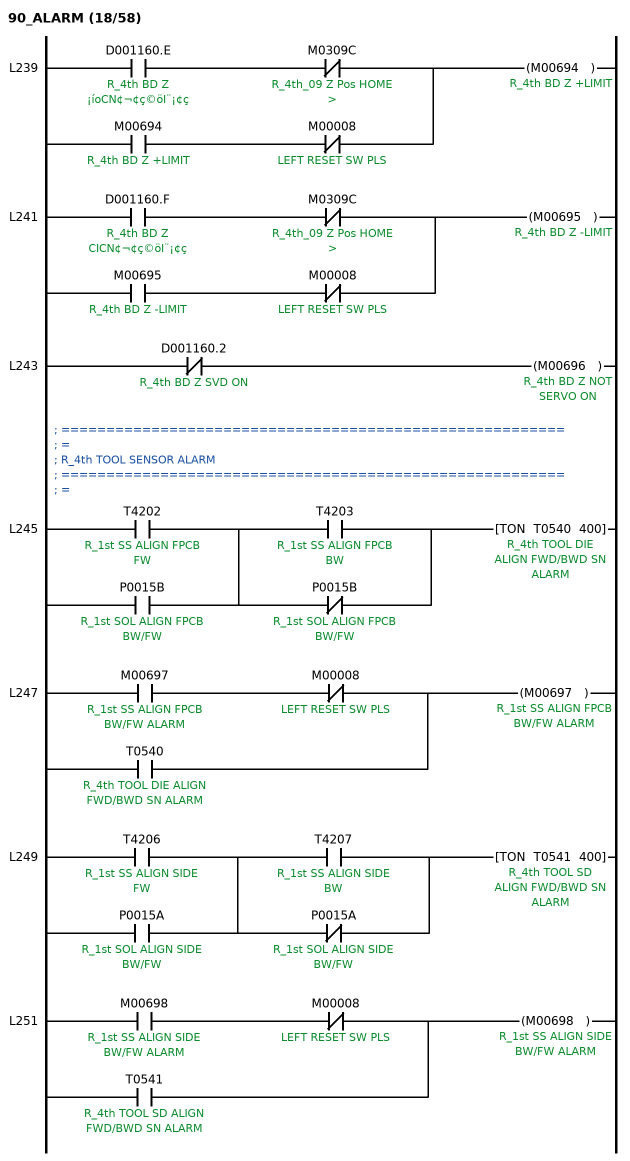
[picture p384: 90_ALARM rungs L239-L251]
; L239
LOAD      D001160.E	// R_4th BD Z ¡íoCN¢¬¢ç©öI¨¡¢ç
AND NOT   M0309C	// R_4th_09 Z Pos HOME >
LOAD      M00694	// R_4th BD Z +LIMIT
AND NOT   M00008	// LEFT RESET SW PLS
OR LOAD
OUT       M00694	// R_4th BD Z +LIMIT
; L241
LOAD      D001160.F	// R_4th BD Z CICN¢¬¢ç©öI¨¡¢ç
AND NOT   M0309C	// R_4th_09 Z Pos HOME >
LOAD      M00695	// R_4th BD Z -LIMIT
AND NOT   M00008	// LEFT RESET SW PLS
OR LOAD
OUT       M00695	// R_4th BD Z -LIMIT
; L243
LOAD NOT  D001160.2	// R_4th BD Z SVD ON
OUT       M00696	// R_4th BD Z NOT SERVO ON
// =========================================================
// 
//        R_4th TOOL SENSOR ALARM
// 
// =========================================================
; L245
LOAD      T4202	// R_1st SS ALIGN FPCB FW
OR        P0015B	// R_1st SOL ALIGN FPCB BW/FW
LOAD      T4203	// R_1st SS ALIGN FPCB BW
OR NOT    P0015B	// R_1st SOL ALIGN FPCB BW/FW
AND LOAD
TON       T0540 400	// R_4th TOOL DIE ALIGN FWD/BWD SN ALARM
; L247
LOAD      M00697	// R_1st SS ALIGN FPCB BW/FW ALARM
AND NOT   M00008	// LEFT RESET SW PLS
OR        T0540	// R_4th TOOL DIE ALIGN FWD/BWD SN ALARM
OUT       M00697	// R_1st SS ALIGN FPCB BW/FW ALARM
; L249
LOAD      T4206	// R_1st SS ALIGN SIDE FW
OR        P0015A	// R_1st SOL ALIGN SIDE BW/FW
LOAD      T4207	// R_1st SS ALIGN SIDE BW
OR NOT    P0015A	// R_1st SOL ALIGN SIDE BW/FW
AND LOAD
TON       T0541 400	// R_4th TOOL SD ALIGN FWD/BWD SN ALARM
; L251
LOAD      M00698	// R_1st SS ALIGN SIDE BW/FW ALARM
AND NOT   M00008	// LEFT RESET SW PLS
OR        T0541	// R_4th TOOL SD ALIGN FWD/BWD SN ALARM
OUT       M00698	// R_1st SS ALIGN SIDE BW/FW ALARM

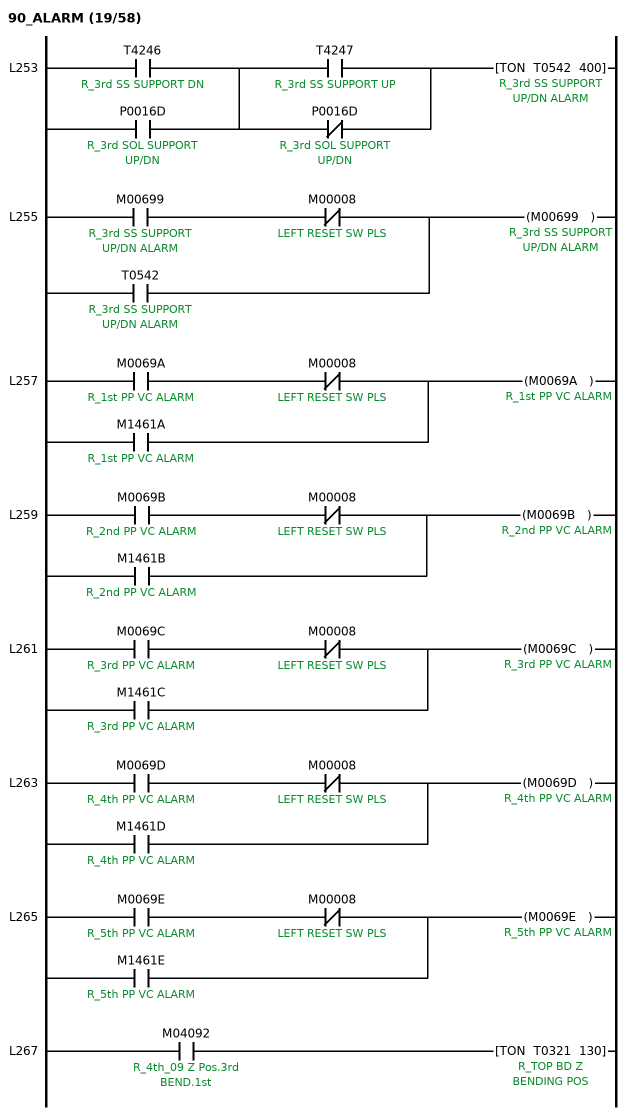
; L253
LOAD      T4246	// R_3rd SS SUPPORT DN
OR        P0016D	// R_3rd SOL SUPPORT UP/DN
LOAD      T4247	// R_3rd SS SUPPORT UP
OR NOT    P0016D	// R_3rd SOL SUPPORT UP/DN
AND LOAD
TON       T0542 400	// R_3rd SS SUPPORT UP/DN ALARM
; L255
LOAD      M00699	// R_3rd SS SUPPORT UP/DN ALARM
AND NOT   M00008	// LEFT RESET SW PLS
OR        T0542	// R_3rd SS SUPPORT UP/DN ALARM
OUT       M00699	// R_3rd SS SUPPORT UP/DN ALARM
; L257
LOAD      M0069A	// R_1st PP VC ALARM
AND NOT   M00008	// LEFT RESET SW PLS
OR        M1461A	// R_1st PP VC ALARM
OUT       M0069A	// R_1st PP VC ALARM
; L259
LOAD      M0069B	// R_2nd PP VC ALARM
AND NOT   M00008	// LEFT RESET SW PLS
OR        M1461B	// R_2nd PP VC ALARM
OUT       M0069B	// R_2nd PP VC ALARM
; L261
LOAD      M0069C	// R_3rd PP VC ALARM
AND NOT   M00008	// LEFT RESET SW PLS
OR        M1461C	// R_3rd PP VC ALARM
OUT       M0069C	// R_3rd PP VC ALARM
; L263
LOAD      M0069D	// R_4th PP VC ALARM
AND NOT   M00008	// LEFT RESET SW PLS
OR        M1461D	// R_4th PP VC ALARM
OUT       M0069D	// R_4th PP VC ALARM
; L265
LOAD      M0069E	// R_5th PP VC ALARM
AND NOT   M00008	// LEFT RESET SW PLS
OR        M1461E	// R_5th PP VC ALARM
OUT       M0069E	// R_5th PP VC ALARM
; L267
LOAD      M04092	// R_4th_09 Z Pos.3rd BEND.1st
TON       T0321 130	// R_TOP BD Z BENDING POS

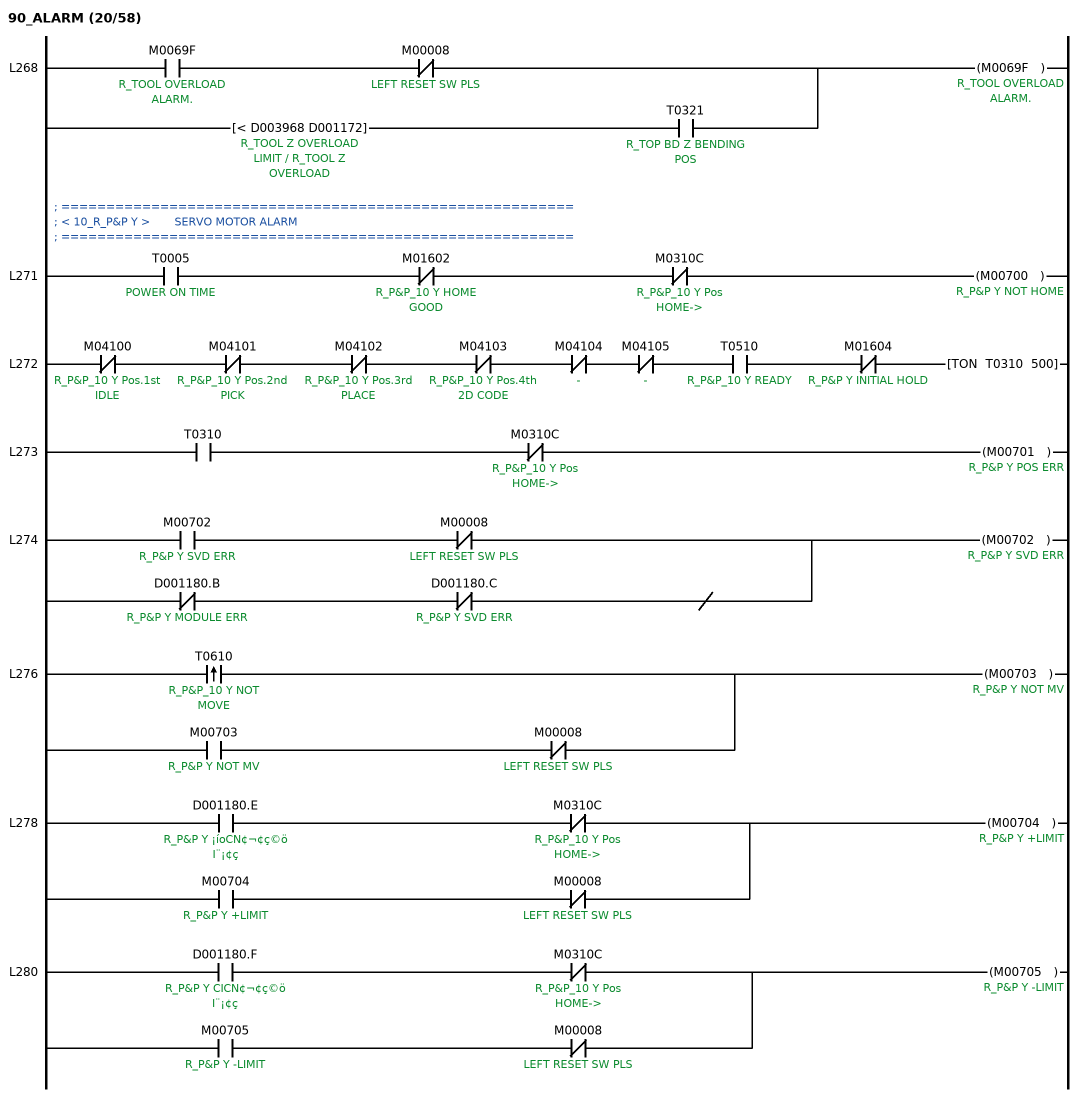
; L268
LOAD      M0069F	// R_TOOL OVERLOAD ALARM.
AND NOT   M00008	// LEFT RESET SW PLS
LOAD<     D003968 D001172	// R_TOOL Z OVERLOAD LIMIT / R_TOOL Z OVERLOAD
AND       T0321	// R_TOP BD Z BENDING POS
OR LOAD
OUT       M0069F	// R_TOOL OVERLOAD ALARM.
// =========================================================
// 
//        < 10_R_P&P Y >       SERVO MOTOR ALARM
// 
// =========================================================
; L271
LOAD      T0005	// POWER ON TIME
AND NOT   M01602	// R_P&P_10 Y HOME GOOD
AND NOT   M0310C	// R_P&P_10 Y Pos HOME->
OUT       M00700	// R_P&P Y NOT HOME
; L272
LOAD NOT  M04100	// R_P&P_10 Y Pos.1st IDLE
AND NOT   M04101	// R_P&P_10 Y Pos.2nd PICK
AND NOT   M04102	// R_P&P_10 Y Pos.3rd PLACE
AND NOT   M04103	// R_P&P_10 Y Pos.4th 2D CODE
AND NOT   M04104	// -
AND NOT   M04105	// -
AND       T0510	// R_P&P_10 Y READY
AND NOT   M01604	// R_P&P Y INITIAL HOLD
TON       T0310 500
; L273
LOAD      T0310
AND NOT   M0310C	// R_P&P_10 Y Pos HOME->
OUT       M00701	// R_P&P Y POS ERR
; L274
LOAD      M00702	// R_P&P Y SVD ERR
AND NOT   M00008	// LEFT RESET SW PLS
LOAD NOT  D001180.B	// R_P&P Y MODULE ERR
AND NOT   D001180.C	// R_P&P Y SVD ERR
NOT
OR LOAD
OUT       M00702	// R_P&P Y SVD ERR
; L276
LOADP     T0610	// R_P&P_10 Y NOT MOVE
LOAD      M00703	// R_P&P Y NOT MV
AND NOT   M00008	// LEFT RESET SW PLS
OR LOAD
OUT       M00703	// R_P&P Y NOT MV
; L278
LOAD      D001180.E	// R_P&P Y ¡íoCN¢¬¢ç©öI¨¡¢ç
AND NOT   M0310C	// R_P&P_10 Y Pos HOME->
LOAD      M00704	// R_P&P Y +LIMIT
AND NOT   M00008	// LEFT RESET SW PLS
OR LOAD
OUT       M00704	// R_P&P Y +LIMIT
; L280
LOAD      D001180.F	// R_P&P Y CICN¢¬¢ç©öI¨¡¢ç
AND NOT   M0310C	// R_P&P_10 Y Pos HOME->
LOAD      M00705	// R_P&P Y -LIMIT
AND NOT   M00008	// LEFT RESET SW PLS
OR LOAD
OUT       M00705	// R_P&P Y -LIMIT

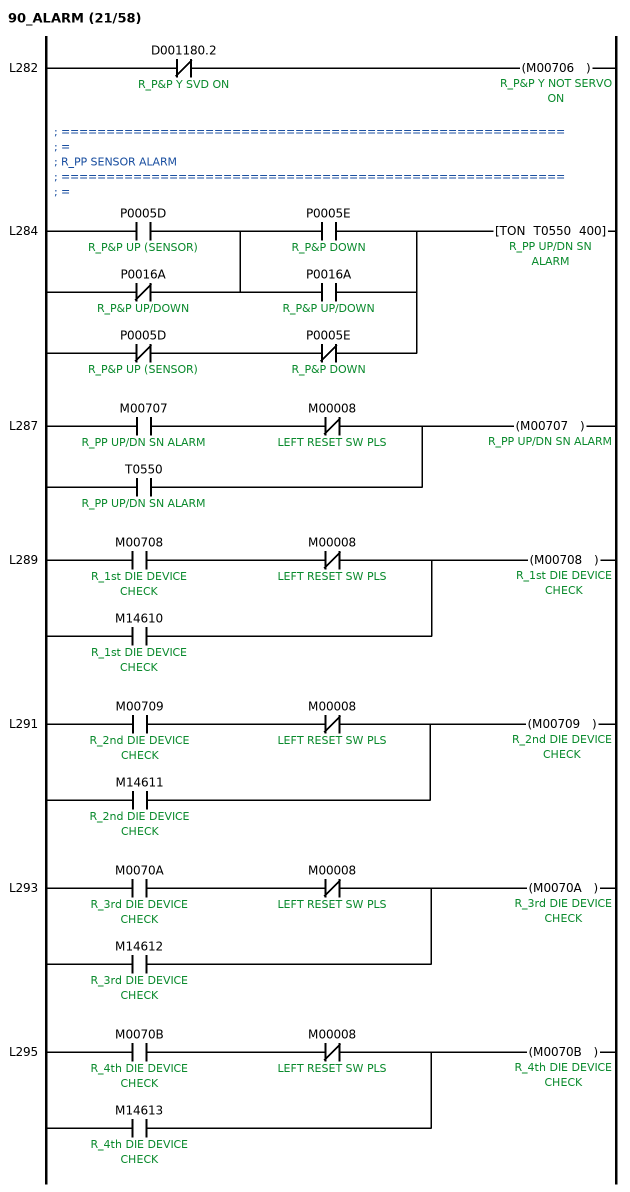
; L282
LOAD NOT  D001180.2	// R_P&P Y SVD ON
OUT       M00706	// R_P&P Y NOT SERVO ON
// =========================================================
// 
//       R_PP SENSOR ALARM
// 
// =========================================================
; L284
LOAD      P0005D	// R_P&P UP (SENSOR)
OR NOT    P0016A	// R_P&P UP/DOWN
LOAD      P0005E	// R_P&P DOWN
OR        P0016A	// R_P&P UP/DOWN
AND LOAD
LOAD NOT  P0005D	// R_P&P UP (SENSOR)
AND NOT   P0005E	// R_P&P DOWN
OR LOAD
TON       T0550 400	// R_PP UP/DN SN ALARM
; L287
LOAD      M00707	// R_PP UP/DN SN ALARM
AND NOT   M00008	// LEFT RESET SW PLS
OR        T0550	// R_PP UP/DN SN ALARM
OUT       M00707	// R_PP UP/DN SN ALARM
; L289
LOAD      M00708	// R_1st DIE DEVICE CHECK
AND NOT   M00008	// LEFT RESET SW PLS
OR        M14610	// R_1st DIE DEVICE CHECK
OUT       M00708	// R_1st DIE DEVICE CHECK
; L291
LOAD      M00709	// R_2nd DIE DEVICE CHECK
AND NOT   M00008	// LEFT RESET SW PLS
OR        M14611	// R_2nd DIE DEVICE CHECK
OUT       M00709	// R_2nd DIE DEVICE CHECK
; L293
LOAD      M0070A	// R_3rd DIE DEVICE CHECK
AND NOT   M00008	// LEFT RESET SW PLS
OR        M14612	// R_3rd DIE DEVICE CHECK
OUT       M0070A	// R_3rd DIE DEVICE CHECK
; L295
LOAD      M0070B	// R_4th DIE DEVICE CHECK
AND NOT   M00008	// LEFT RESET SW PLS
OR        M14613	// R_4th DIE DEVICE CHECK
OUT       M0070B	// R_4th DIE DEVICE CHECK

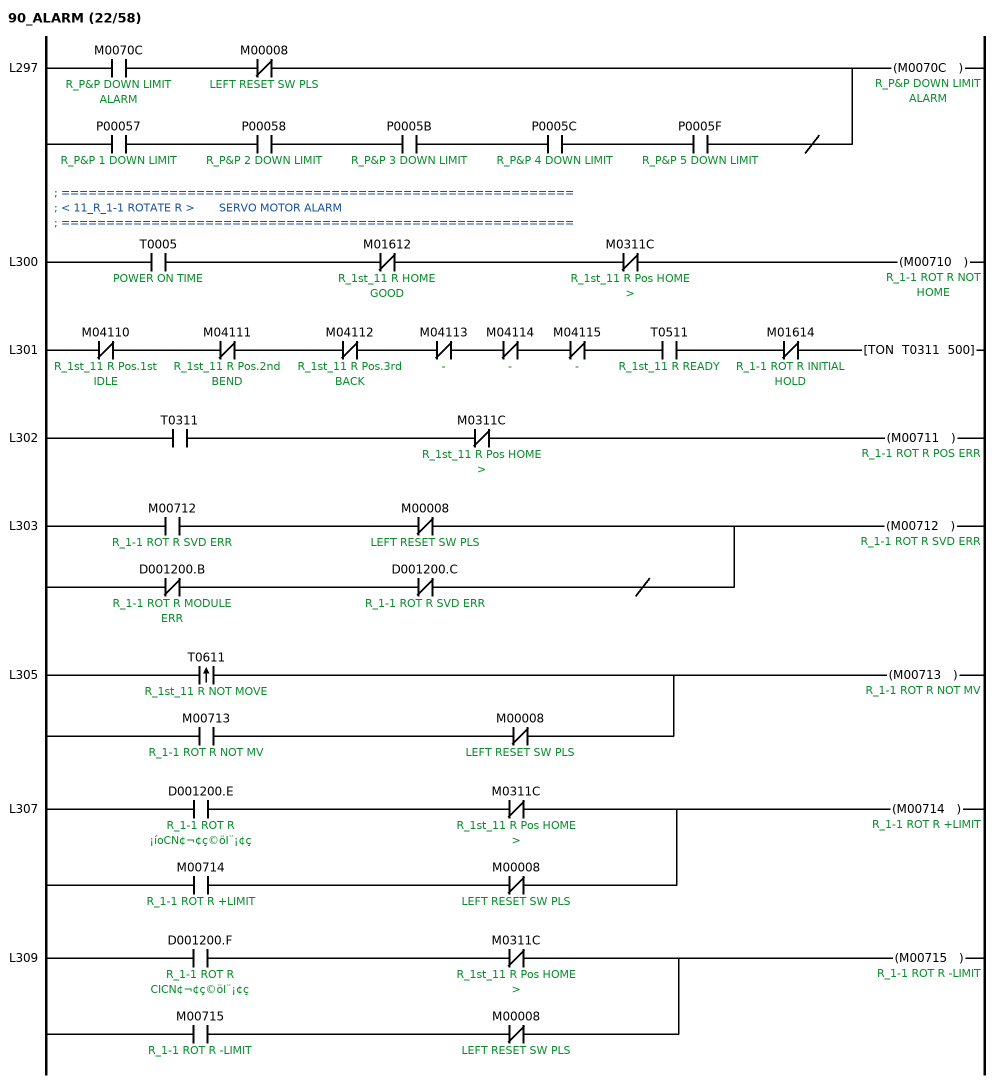
; L297
LOAD      M0070C	// R_P&P DOWN LIMIT ALARM
AND NOT   M00008	// LEFT RESET SW PLS
LOAD      P00057	// R_P&P 1 DOWN LIMIT
AND       P00058	// R_P&P 2 DOWN LIMIT
AND       P0005B	// R_P&P 3 DOWN LIMIT
AND       P0005C	// R_P&P 4 DOWN LIMIT
AND       P0005F	// R_P&P 5 DOWN LIMIT
NOT
OR LOAD
OUT       M0070C	// R_P&P DOWN LIMIT ALARM
// =========================================================
// 
//        < 11_R_1-1 ROTATE R >       SERVO MOTOR ALARM
// 
// =========================================================
; L300
LOAD      T0005	// POWER ON TIME
AND NOT   M01612	// R_1st_11 R HOME GOOD
AND NOT   M0311C	// R_1st_11 R Pos HOME >
OUT       M00710	// R_1-1 ROT R NOT HOME
; L301
LOAD NOT  M04110	// R_1st_11 R Pos.1st IDLE
AND NOT   M04111	// R_1st_11 R Pos.2nd BEND
AND NOT   M04112	// R_1st_11 R Pos.3rd BACK
AND NOT   M04113	// -
AND NOT   M04114	// -
AND NOT   M04115	// -
AND       T0511	// R_1st_11 R READY
AND NOT   M01614	// R_1-1 ROT R INITIAL HOLD
TON       T0311 500
; L302
LOAD      T0311
AND NOT   M0311C	// R_1st_11 R Pos HOME >
OUT       M00711	// R_1-1 ROT R POS ERR
; L303
LOAD      M00712	// R_1-1 ROT R SVD ERR
AND NOT   M00008	// LEFT RESET SW PLS
LOAD NOT  D001200.B	// R_1-1 ROT R MODULE ERR
AND NOT   D001200.C	// R_1-1 ROT R SVD ERR
NOT
OR LOAD
OUT       M00712	// R_1-1 ROT R SVD ERR
; L305
LOADP     T0611	// R_1st_11 R NOT MOVE
LOAD      M00713	// R_1-1 ROT R NOT MV
AND NOT   M00008	// LEFT RESET SW PLS
OR LOAD
OUT       M00713	// R_1-1 ROT R NOT MV
; L307
LOAD      D001200.E	// R_1-1 ROT R ¡íoCN¢¬¢ç©öI¨¡¢ç
AND NOT   M0311C	// R_1st_11 R Pos HOME >
LOAD      M00714	// R_1-1 ROT R +LIMIT
AND NOT   M00008	// LEFT RESET SW PLS
OR LOAD
OUT       M00714	// R_1-1 ROT R +LIMIT
; L309
LOAD      D001200.F	// R_1-1 ROT R CICN¢¬¢ç©öI¨¡¢ç
AND NOT   M0311C	// R_1st_11 R Pos HOME >
LOAD      M00715	// R_1-1 ROT R -LIMIT
AND NOT   M00008	// LEFT RESET SW PLS
OR LOAD
OUT       M00715	// R_1-1 ROT R -LIMIT

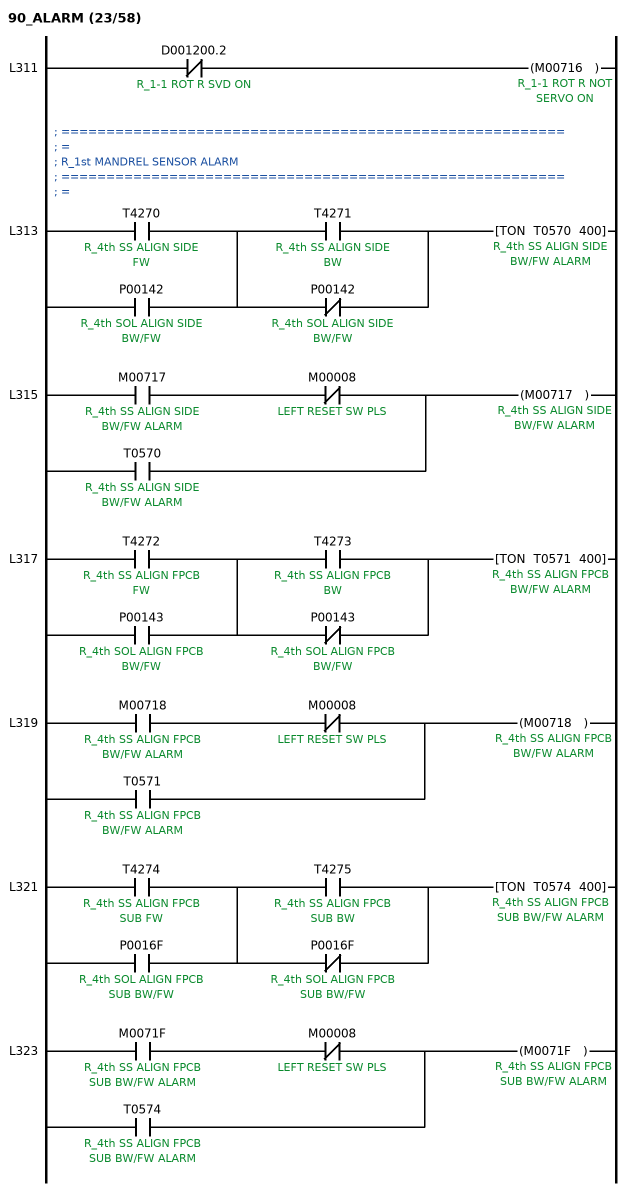
; L311
LOAD NOT  D001200.2	// R_1-1 ROT R SVD ON
OUT       M00716	// R_1-1 ROT R NOT SERVO ON
// =========================================================
// 
//        R_1st MANDREL SENSOR ALARM
// 
// =========================================================
; L313
LOAD      T4270	// R_4th SS ALIGN SIDE FW
OR        P00142	// R_4th SOL ALIGN SIDE BW/FW
LOAD      T4271	// R_4th SS ALIGN SIDE BW
OR NOT    P00142	// R_4th SOL ALIGN SIDE BW/FW
AND LOAD
TON       T0570 400	// R_4th SS ALIGN SIDE BW/FW ALARM
; L315
LOAD      M00717	// R_4th SS ALIGN SIDE BW/FW ALARM
AND NOT   M00008	// LEFT RESET SW PLS
OR        T0570	// R_4th SS ALIGN SIDE BW/FW ALARM
OUT       M00717	// R_4th SS ALIGN SIDE BW/FW ALARM
; L317
LOAD      T4272	// R_4th SS ALIGN FPCB FW
OR        P00143	// R_4th SOL ALIGN FPCB BW/FW
LOAD      T4273	// R_4th SS ALIGN FPCB BW
OR NOT    P00143	// R_4th SOL ALIGN FPCB BW/FW
AND LOAD
TON       T0571 400	// R_4th SS ALIGN FPCB BW/FW ALARM
; L319
LOAD      M00718	// R_4th SS ALIGN FPCB BW/FW ALARM
AND NOT   M00008	// LEFT RESET SW PLS
OR        T0571	// R_4th SS ALIGN FPCB BW/FW ALARM
OUT       M00718	// R_4th SS ALIGN FPCB BW/FW ALARM
; L321
LOAD      T4274	// R_4th SS ALIGN FPCB SUB FW
OR        P0016F	// R_4th SOL ALIGN FPCB SUB BW/FW
LOAD      T4275	// R_4th SS ALIGN FPCB SUB BW
OR NOT    P0016F	// R_4th SOL ALIGN FPCB SUB BW/FW
AND LOAD
TON       T0574 400	// R_4th SS ALIGN FPCB SUB BW/FW ALARM
; L323
LOAD      M0071F	// R_4th SS ALIGN FPCB SUB BW/FW ALARM
AND NOT   M00008	// LEFT RESET SW PLS
OR        T0574	// R_4th SS ALIGN FPCB SUB BW/FW ALARM
OUT       M0071F	// R_4th SS ALIGN FPCB SUB BW/FW ALARM

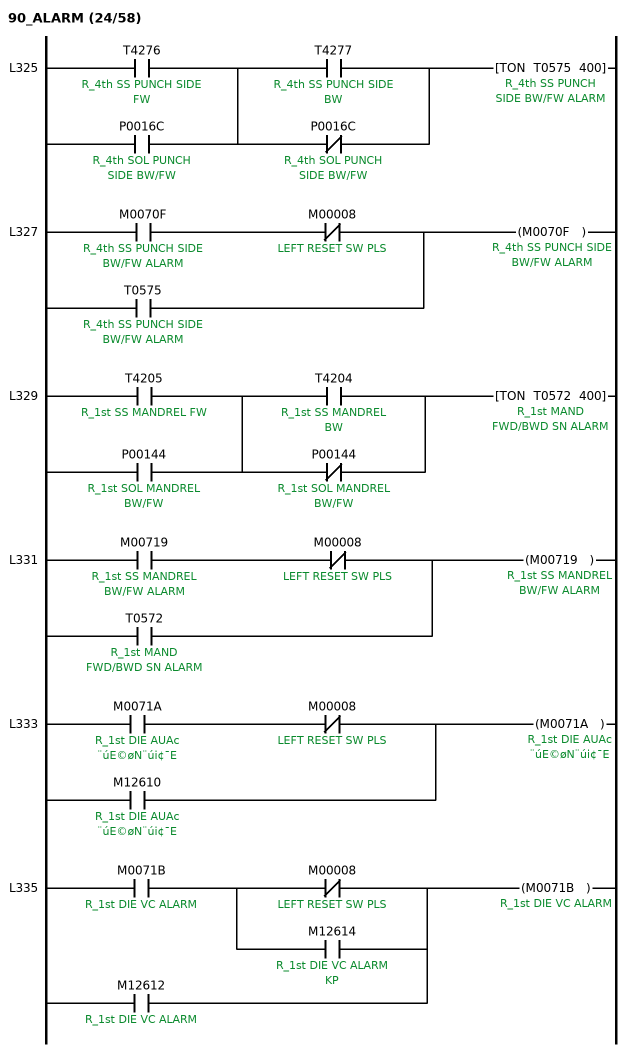
; L325
LOAD      T4276	// R_4th SS PUNCH SIDE FW
OR        P0016C	// R_4th SOL PUNCH SIDE BW/FW
LOAD      T4277	// R_4th SS PUNCH SIDE BW
OR NOT    P0016C	// R_4th SOL PUNCH SIDE BW/FW
AND LOAD
TON       T0575 400	// R_4th SS PUNCH SIDE BW/FW ALARM
; L327
LOAD      M0070F	// R_4th SS PUNCH SIDE BW/FW ALARM
AND NOT   M00008	// LEFT RESET SW PLS
OR        T0575	// R_4th SS PUNCH SIDE BW/FW ALARM
OUT       M0070F	// R_4th SS PUNCH SIDE BW/FW ALARM
; L329
LOAD      T4205	// R_1st SS MANDREL FW
OR        P00144	// R_1st SOL MANDREL BW/FW
LOAD      T4204	// R_1st SS MANDREL BW
OR NOT    P00144	// R_1st SOL MANDREL BW/FW
AND LOAD
TON       T0572 400	// R_1st MAND FWD/BWD SN ALARM
; L331
LOAD      M00719	// R_1st SS MANDREL BW/FW ALARM
AND NOT   M00008	// LEFT RESET SW PLS
OR        T0572	// R_1st MAND FWD/BWD SN ALARM
OUT       M00719	// R_1st SS MANDREL BW/FW ALARM
; L333
LOAD      M0071A	// R_1st DIE AUAc ¨úE©øN¨úi¢¯E
AND NOT   M00008	// LEFT RESET SW PLS
OR        M12610	// R_1st DIE AUAc ¨úE©øN¨úi¢¯E
OUT       M0071A	// R_1st DIE AUAc ¨úE©øN¨úi¢¯E
; L335
LOAD      M0071B	// R_1st DIE VC ALARM
LOAD NOT  M00008	// LEFT RESET SW PLS
OR        M12614	// R_1st DIE VC ALARM KP
AND LOAD
OR        M12612	// R_1st DIE VC ALARM
OUT       M0071B	// R_1st DIE VC ALARM

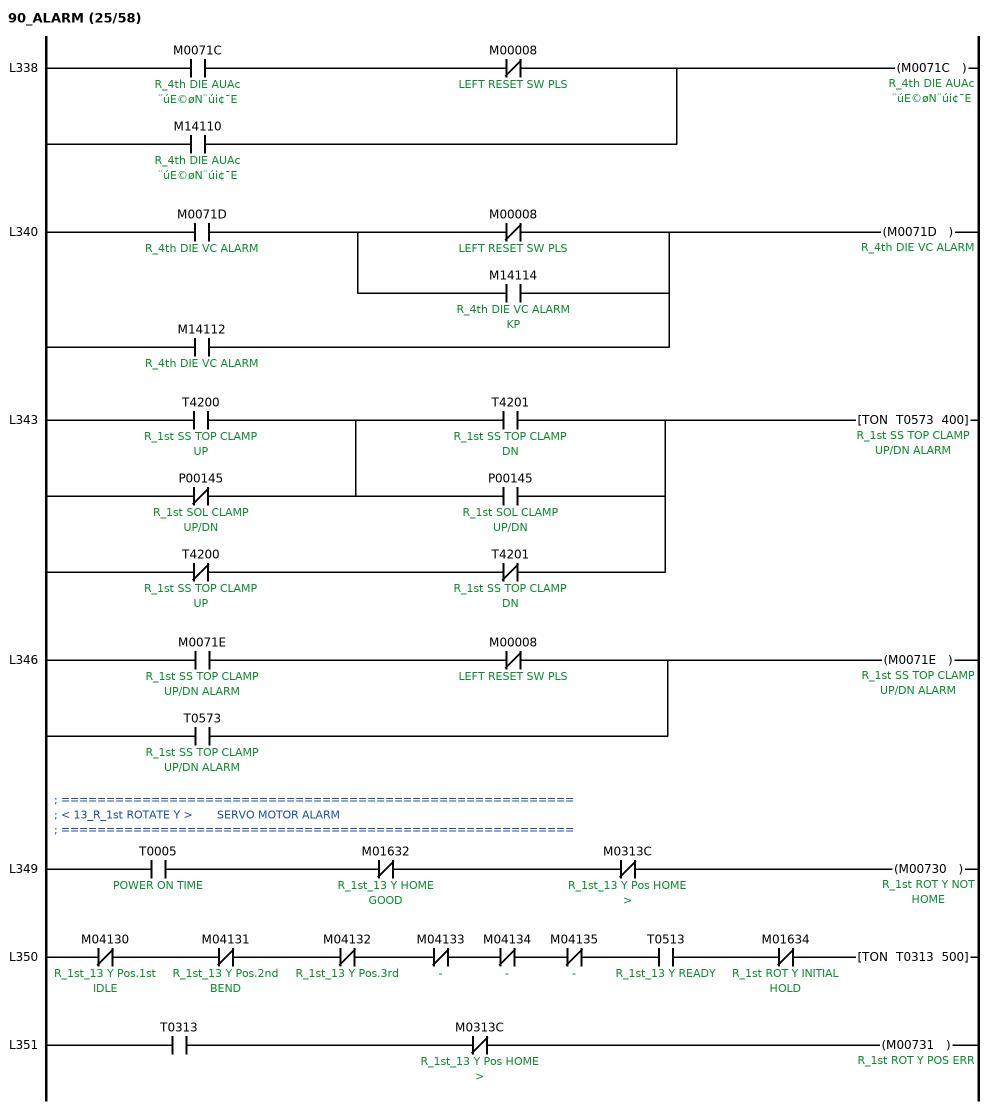
; L338
LOAD      M0071C	// R_4th DIE AUAc ¨úE©øN¨úi¢¯E
AND NOT   M00008	// LEFT RESET SW PLS
OR        M14110	// R_4th DIE AUAc ¨úE©øN¨úi¢¯E
OUT       M0071C	// R_4th DIE AUAc ¨úE©øN¨úi¢¯E
; L340
LOAD      M0071D	// R_4th DIE VC ALARM
LOAD NOT  M00008	// LEFT RESET SW PLS
OR        M14114	// R_4th DIE VC ALARM KP
AND LOAD
OR        M14112	// R_4th DIE VC ALARM
OUT       M0071D	// R_4th DIE VC ALARM
; L343
LOAD      T4200	// R_1st SS TOP CLAMP UP
OR NOT    P00145	// R_1st SOL CLAMP UP/DN
LOAD      T4201	// R_1st SS TOP CLAMP DN
OR        P00145	// R_1st SOL CLAMP UP/DN
AND LOAD
LOAD NOT  T4200	// R_1st SS TOP CLAMP UP
AND NOT   T4201	// R_1st SS TOP CLAMP DN
OR LOAD
TON       T0573 400	// R_1st SS TOP CLAMP UP/DN ALARM
; L346
LOAD      M0071E	// R_1st SS TOP CLAMP UP/DN ALARM
AND NOT   M00008	// LEFT RESET SW PLS
OR        T0573	// R_1st SS TOP CLAMP UP/DN ALARM
OUT       M0071E	// R_1st SS TOP CLAMP UP/DN ALARM
// =========================================================
// 
//        < 13_R_1st ROTATE Y >       SERVO MOTOR ALARM
// 
// =========================================================
; L349
LOAD      T0005	// POWER ON TIME
AND NOT   M01632	// R_1st_13 Y HOME GOOD
AND NOT   M0313C	// R_1st_13 Y Pos HOME >
OUT       M00730	// R_1st ROT Y NOT HOME
; L350
LOAD NOT  M04130	// R_1st_13 Y Pos.1st IDLE
AND NOT   M04131	// R_1st_13 Y Pos.2nd BEND
AND NOT   M04132	// R_1st_13 Y Pos.3rd
AND NOT   M04133	// -
AND NOT   M04134	// -
AND NOT   M04135	// -
AND       T0513	// R_1st_13 Y READY
AND NOT   M01634	// R_1st ROT Y INITIAL HOLD
TON       T0313 500
; L351
LOAD      T0313
AND NOT   M0313C	// R_1st_13 Y Pos HOME >
OUT       M00731	// R_1st ROT Y POS ERR

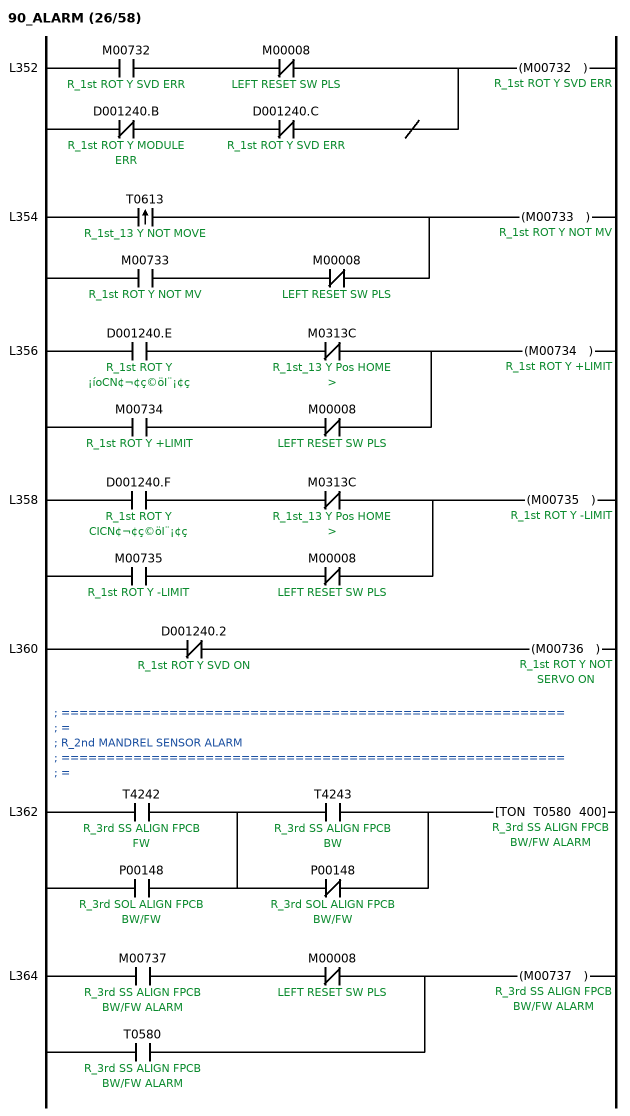
; L352
LOAD      M00732	// R_1st ROT Y SVD ERR
AND NOT   M00008	// LEFT RESET SW PLS
LOAD NOT  D001240.B	// R_1st ROT Y MODULE ERR
AND NOT   D001240.C	// R_1st ROT Y SVD ERR
NOT
OR LOAD
OUT       M00732	// R_1st ROT Y SVD ERR
; L354
LOADP     T0613	// R_1st_13 Y NOT MOVE
LOAD      M00733	// R_1st ROT Y NOT MV
AND NOT   M00008	// LEFT RESET SW PLS
OR LOAD
OUT       M00733	// R_1st ROT Y NOT MV
; L356
LOAD      D001240.E	// R_1st ROT Y ¡íoCN¢¬¢ç©öI¨¡¢ç
AND NOT   M0313C	// R_1st_13 Y Pos HOME >
LOAD      M00734	// R_1st ROT Y +LIMIT
AND NOT   M00008	// LEFT RESET SW PLS
OR LOAD
OUT       M00734	// R_1st ROT Y +LIMIT
; L358
LOAD      D001240.F	// R_1st ROT Y CICN¢¬¢ç©öI¨¡¢ç
AND NOT   M0313C	// R_1st_13 Y Pos HOME >
LOAD      M00735	// R_1st ROT Y -LIMIT
AND NOT   M00008	// LEFT RESET SW PLS
OR LOAD
OUT       M00735	// R_1st ROT Y -LIMIT
; L360
LOAD NOT  D001240.2	// R_1st ROT Y SVD ON
OUT       M00736	// R_1st ROT Y NOT SERVO ON
// =========================================================
// 
//        R_2nd MANDREL SENSOR ALARM
// 
// =========================================================
; L362
LOAD      T4242	// R_3rd SS ALIGN FPCB FW
OR        P00148	// R_3rd SOL ALIGN FPCB BW/FW
LOAD      T4243	// R_3rd SS ALIGN FPCB BW
OR NOT    P00148	// R_3rd SOL ALIGN FPCB BW/FW
AND LOAD
TON       T0580 400	// R_3rd SS ALIGN FPCB BW/FW ALARM
; L364
LOAD      M00737	// R_3rd SS ALIGN FPCB BW/FW ALARM
AND NOT   M00008	// LEFT RESET SW PLS
OR        T0580	// R_3rd SS ALIGN FPCB BW/FW ALARM
OUT       M00737	// R_3rd SS ALIGN FPCB BW/FW ALARM

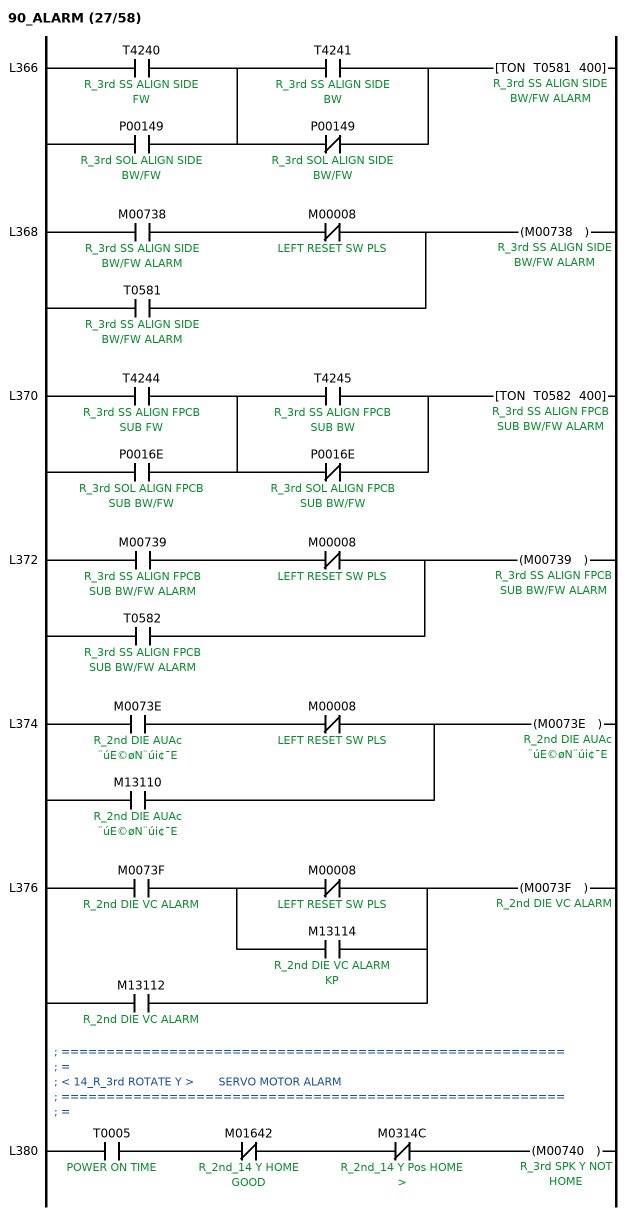
; L366
LOAD      T4240	// R_3rd SS ALIGN SIDE FW
OR        P00149	// R_3rd SOL ALIGN SIDE BW/FW
LOAD      T4241	// R_3rd SS ALIGN SIDE BW
OR NOT    P00149	// R_3rd SOL ALIGN SIDE BW/FW
AND LOAD
TON       T0581 400	// R_3rd SS ALIGN SIDE BW/FW ALARM
; L368
LOAD      M00738	// R_3rd SS ALIGN SIDE BW/FW ALARM
AND NOT   M00008	// LEFT RESET SW PLS
OR        T0581	// R_3rd SS ALIGN SIDE BW/FW ALARM
OUT       M00738	// R_3rd SS ALIGN SIDE BW/FW ALARM
; L370
LOAD      T4244	// R_3rd SS ALIGN FPCB SUB FW
OR        P0016E	// R_3rd SOL ALIGN FPCB SUB BW/FW
LOAD      T4245	// R_3rd SS ALIGN FPCB SUB BW
OR NOT    P0016E	// R_3rd SOL ALIGN FPCB SUB BW/FW
AND LOAD
TON       T0582 400	// R_3rd SS ALIGN FPCB SUB BW/FW ALARM
; L372
LOAD      M00739	// R_3rd SS ALIGN FPCB SUB BW/FW ALARM
AND NOT   M00008	// LEFT RESET SW PLS
OR        T0582	// R_3rd SS ALIGN FPCB SUB BW/FW ALARM
OUT       M00739	// R_3rd SS ALIGN FPCB SUB BW/FW ALARM
; L374
LOAD      M0073E	// R_2nd DIE AUAc ¨úE©øN¨úi¢¯E
AND NOT   M00008	// LEFT RESET SW PLS
OR        M13110	// R_2nd DIE AUAc ¨úE©øN¨úi¢¯E
OUT       M0073E	// R_2nd DIE AUAc ¨úE©øN¨úi¢¯E
; L376
LOAD      M0073F	// R_2nd DIE VC ALARM
LOAD NOT  M00008	// LEFT RESET SW PLS
OR        M13114	// R_2nd DIE VC ALARM KP
AND LOAD
OR        M13112	// R_2nd DIE VC ALARM
OUT       M0073F	// R_2nd DIE VC ALARM
// =========================================================
// 
//        < 14_R_3rd ROTATE Y >       SERVO MOTOR ALARM
// 
// =========================================================
; L380
LOAD      T0005	// POWER ON TIME
AND NOT   M01642	// R_2nd_14 Y HOME GOOD
AND NOT   M0314C	// R_2nd_14 Y Pos HOME >
OUT       M00740	// R_3rd SPK Y NOT HOME

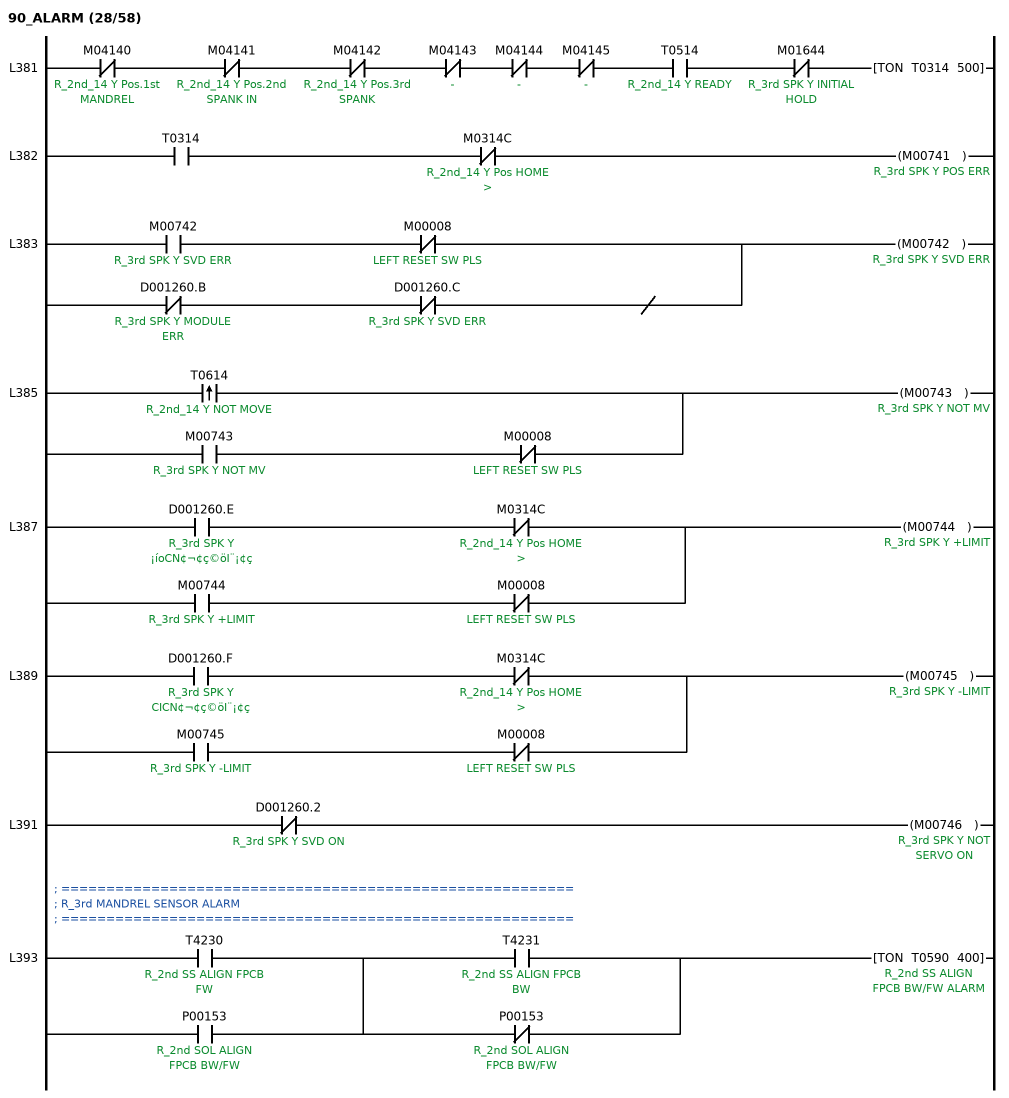
; L381
LOAD NOT  M04140	// R_2nd_14 Y Pos.1st MANDREL
AND NOT   M04141	// R_2nd_14 Y Pos.2nd SPANK IN
AND NOT   M04142	// R_2nd_14 Y Pos.3rd SPANK
AND NOT   M04143	// -
AND NOT   M04144	// -
AND NOT   M04145	// -
AND       T0514	// R_2nd_14 Y READY
AND NOT   M01644	// R_3rd SPK Y INITIAL HOLD
TON       T0314 500
; L382
LOAD      T0314
AND NOT   M0314C	// R_2nd_14 Y Pos HOME >
OUT       M00741	// R_3rd SPK Y POS ERR
; L383
LOAD      M00742	// R_3rd SPK Y SVD ERR
AND NOT   M00008	// LEFT RESET SW PLS
LOAD NOT  D001260.B	// R_3rd SPK Y MODULE ERR
AND NOT   D001260.C	// R_3rd SPK Y SVD ERR
NOT
OR LOAD
OUT       M00742	// R_3rd SPK Y SVD ERR
; L385
LOADP     T0614	// R_2nd_14 Y NOT MOVE
LOAD      M00743	// R_3rd SPK Y NOT MV
AND NOT   M00008	// LEFT RESET SW PLS
OR LOAD
OUT       M00743	// R_3rd SPK Y NOT MV
; L387
LOAD      D001260.E	// R_3rd SPK Y ¡íoCN¢¬¢ç©öI¨¡¢ç
AND NOT   M0314C	// R_2nd_14 Y Pos HOME >
LOAD      M00744	// R_3rd SPK Y +LIMIT
AND NOT   M00008	// LEFT RESET SW PLS
OR LOAD
OUT       M00744	// R_3rd SPK Y +LIMIT
; L389
LOAD      D001260.F	// R_3rd SPK Y CICN¢¬¢ç©öI¨¡¢ç
AND NOT   M0314C	// R_2nd_14 Y Pos HOME >
LOAD      M00745	// R_3rd SPK Y -LIMIT
AND NOT   M00008	// LEFT RESET SW PLS
OR LOAD
OUT       M00745	// R_3rd SPK Y -LIMIT
; L391
LOAD NOT  D001260.2	// R_3rd SPK Y SVD ON
OUT       M00746	// R_3rd SPK Y NOT SERVO ON
// =========================================================
// 
//        R_3rd MANDREL SENSOR ALARM
// 
// =========================================================
; L393
LOAD      T4230	// R_2nd SS ALIGN FPCB FW
OR        P00153	// R_2nd SOL ALIGN FPCB BW/FW
LOAD      T4231	// R_2nd SS ALIGN FPCB BW
OR NOT    P00153	// R_2nd SOL ALIGN FPCB BW/FW
AND LOAD
TON       T0590 400	// R_2nd SS ALIGN FPCB BW/FW ALARM

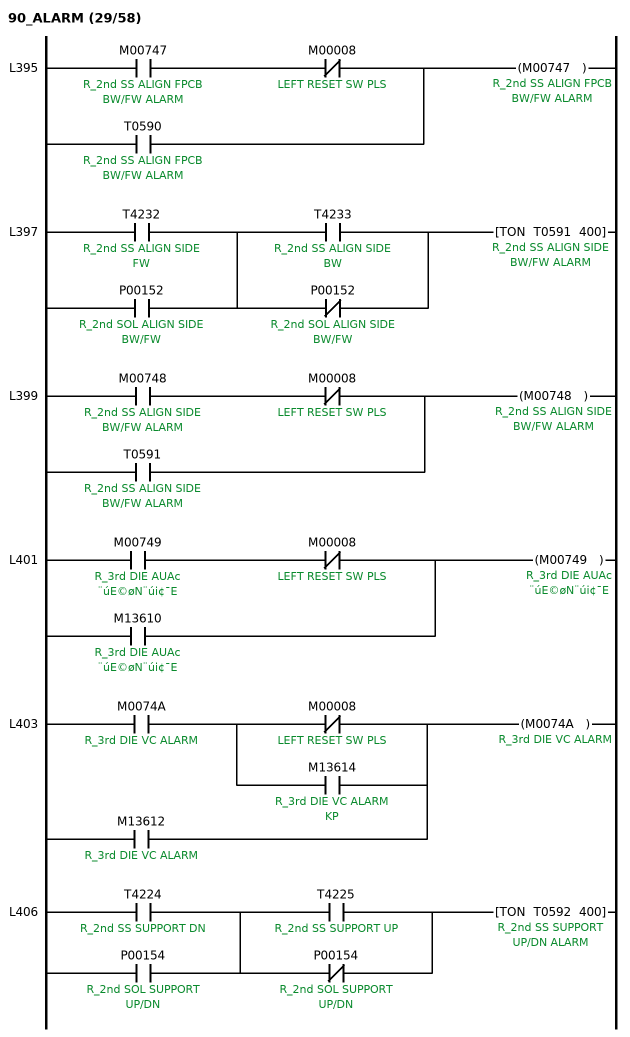
; L395
LOAD      M00747	// R_2nd SS ALIGN FPCB BW/FW ALARM
AND NOT   M00008	// LEFT RESET SW PLS
OR        T0590	// R_2nd SS ALIGN FPCB BW/FW ALARM
OUT       M00747	// R_2nd SS ALIGN FPCB BW/FW ALARM
; L397
LOAD      T4232	// R_2nd SS ALIGN SIDE FW
OR        P00152	// R_2nd SOL ALIGN SIDE BW/FW
LOAD      T4233	// R_2nd SS ALIGN SIDE BW
OR NOT    P00152	// R_2nd SOL ALIGN SIDE BW/FW
AND LOAD
TON       T0591 400	// R_2nd SS ALIGN SIDE BW/FW ALARM
; L399
LOAD      M00748	// R_2nd SS ALIGN SIDE BW/FW ALARM
AND NOT   M00008	// LEFT RESET SW PLS
OR        T0591	// R_2nd SS ALIGN SIDE BW/FW ALARM
OUT       M00748	// R_2nd SS ALIGN SIDE BW/FW ALARM
; L401
LOAD      M00749	// R_3rd DIE AUAc ¨úE©øN¨úi¢¯E
AND NOT   M00008	// LEFT RESET SW PLS
OR        M13610	// R_3rd DIE AUAc ¨úE©øN¨úi¢¯E
OUT       M00749	// R_3rd DIE AUAc ¨úE©øN¨úi¢¯E
; L403
LOAD      M0074A	// R_3rd DIE VC ALARM
LOAD NOT  M00008	// LEFT RESET SW PLS
OR        M13614	// R_3rd DIE VC ALARM KP
AND LOAD
OR        M13612	// R_3rd DIE VC ALARM
OUT       M0074A	// R_3rd DIE VC ALARM
; L406
LOAD      T4224	// R_2nd SS SUPPORT DN
OR        P00154	// R_2nd SOL SUPPORT UP/DN
LOAD      T4225	// R_2nd SS SUPPORT UP
OR NOT    P00154	// R_2nd SOL SUPPORT UP/DN
AND LOAD
TON       T0592 400	// R_2nd SS SUPPORT UP/DN ALARM

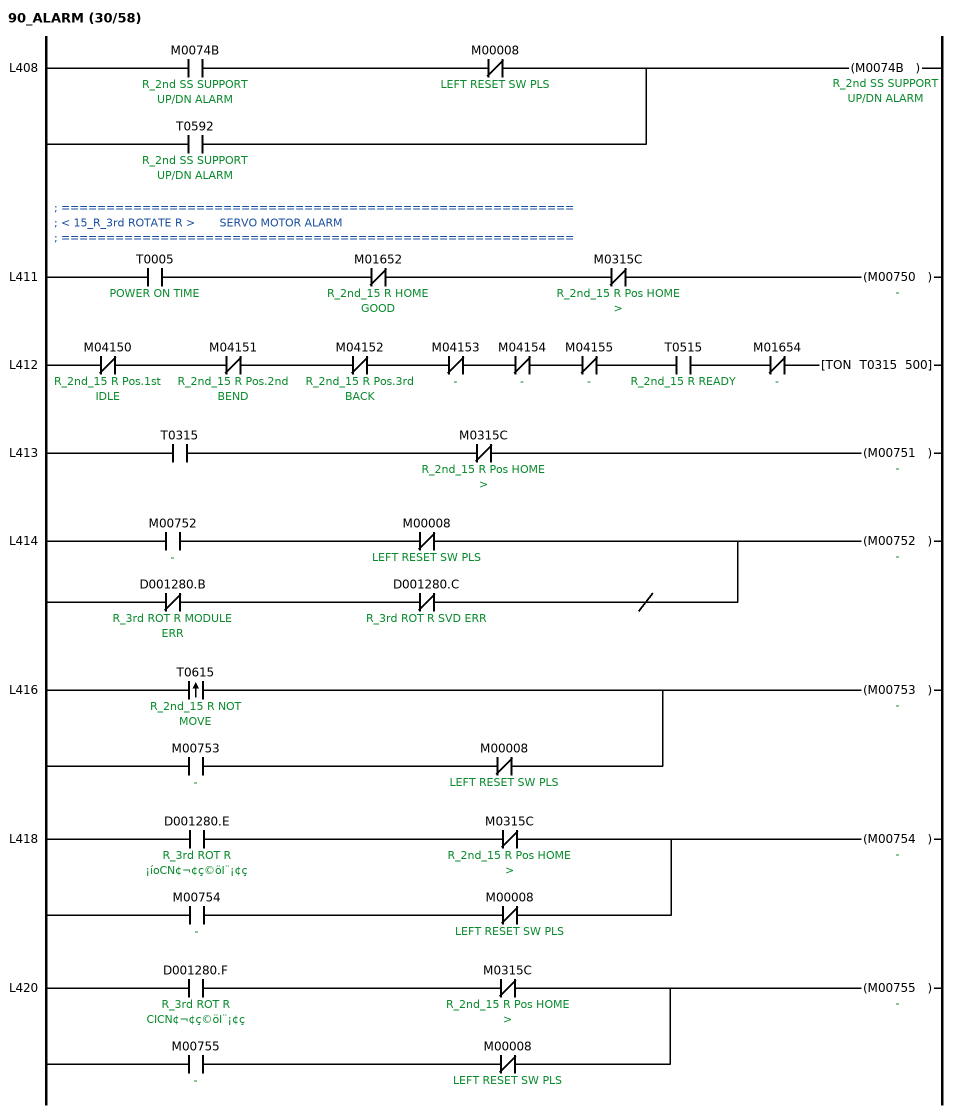
; L408
LOAD      M0074B	// R_2nd SS SUPPORT UP/DN ALARM
AND NOT   M00008	// LEFT RESET SW PLS
OR        T0592	// R_2nd SS SUPPORT UP/DN ALARM
OUT       M0074B	// R_2nd SS SUPPORT UP/DN ALARM
// =========================================================
// 
//        < 15_R_3rd ROTATE R >       SERVO MOTOR ALARM
// 
// =========================================================
; L411
LOAD      T0005	// POWER ON TIME
AND NOT   M01652	// R_2nd_15 R HOME GOOD
AND NOT   M0315C	// R_2nd_15 R Pos HOME >
OUT       M00750	// -
; L412
LOAD NOT  M04150	// R_2nd_15 R Pos.1st IDLE
AND NOT   M04151	// R_2nd_15 R Pos.2nd BEND
AND NOT   M04152	// R_2nd_15 R Pos.3rd BACK
AND NOT   M04153	// -
AND NOT   M04154	// -
AND NOT   M04155	// -
AND       T0515	// R_2nd_15 R READY
AND NOT   M01654	// -
TON       T0315 500
; L413
LOAD      T0315
AND NOT   M0315C	// R_2nd_15 R Pos HOME >
OUT       M00751	// -
; L414
LOAD      M00752	// -
AND NOT   M00008	// LEFT RESET SW PLS
LOAD NOT  D001280.B	// R_3rd ROT R MODULE ERR
AND NOT   D001280.C	// R_3rd ROT R SVD ERR
NOT
OR LOAD
OUT       M00752	// -
; L416
LOADP     T0615	// R_2nd_15 R NOT MOVE
LOAD      M00753	// -
AND NOT   M00008	// LEFT RESET SW PLS
OR LOAD
OUT       M00753	// -
; L418
LOAD      D001280.E	// R_3rd ROT R ¡íoCN¢¬¢ç©öI¨¡¢ç
AND NOT   M0315C	// R_2nd_15 R Pos HOME >
LOAD      M00754	// -
AND NOT   M00008	// LEFT RESET SW PLS
OR LOAD
OUT       M00754	// -
; L420
LOAD      D001280.F	// R_3rd ROT R CICN¢¬¢ç©öI¨¡¢ç
AND NOT   M0315C	// R_2nd_15 R Pos HOME >
LOAD      M00755	// -
AND NOT   M00008	// LEFT RESET SW PLS
OR LOAD
OUT       M00755	// -

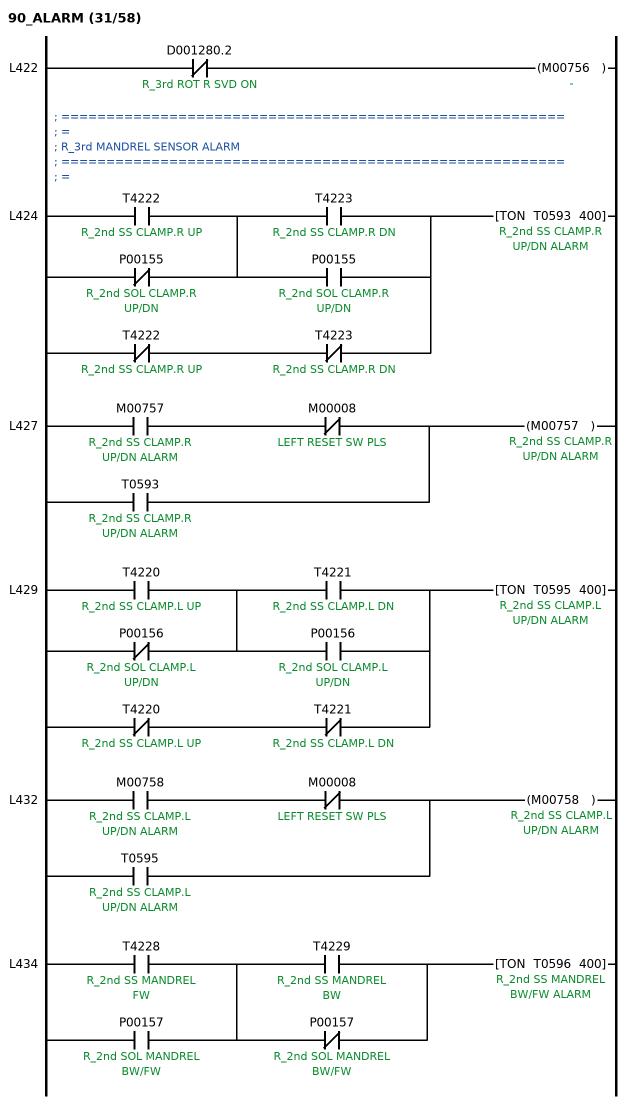
; L422
LOAD NOT  D001280.2	// R_3rd ROT R SVD ON
OUT       M00756	// -
// =========================================================
// 
//        R_3rd MANDREL SENSOR ALARM
// 
// =========================================================
; L424
LOAD      T4222	// R_2nd SS CLAMP.R UP
OR NOT    P00155	// R_2nd SOL CLAMP.R UP/DN
LOAD      T4223	// R_2nd SS CLAMP.R DN
OR        P00155	// R_2nd SOL CLAMP.R UP/DN
AND LOAD
LOAD NOT  T4222	// R_2nd SS CLAMP.R UP
AND NOT   T4223	// R_2nd SS CLAMP.R DN
OR LOAD
TON       T0593 400	// R_2nd SS CLAMP.R UP/DN ALARM
; L427
LOAD      M00757	// R_2nd SS CLAMP.R UP/DN ALARM
AND NOT   M00008	// LEFT RESET SW PLS
OR        T0593	// R_2nd SS CLAMP.R UP/DN ALARM
OUT       M00757	// R_2nd SS CLAMP.R UP/DN ALARM
; L429
LOAD      T4220	// R_2nd SS CLAMP.L UP
OR NOT    P00156	// R_2nd SOL CLAMP.L UP/DN
LOAD      T4221	// R_2nd SS CLAMP.L DN
OR        P00156	// R_2nd SOL CLAMP.L UP/DN
AND LOAD
LOAD NOT  T4220	// R_2nd SS CLAMP.L UP
AND NOT   T4221	// R_2nd SS CLAMP.L DN
OR LOAD
TON       T0595 400	// R_2nd SS CLAMP.L UP/DN ALARM
; L432
LOAD      M00758	// R_2nd SS CLAMP.L UP/DN ALARM
AND NOT   M00008	// LEFT RESET SW PLS
OR        T0595	// R_2nd SS CLAMP.L UP/DN ALARM
OUT       M00758	// R_2nd SS CLAMP.L UP/DN ALARM
; L434
LOAD      T4228	// R_2nd SS MANDREL FW
OR        P00157	// R_2nd SOL MANDREL BW/FW
LOAD      T4229	// R_2nd SS MANDREL BW
OR NOT    P00157	// R_2nd SOL MANDREL BW/FW
AND LOAD
TON       T0596 400	// R_2nd SS MANDREL BW/FW ALARM

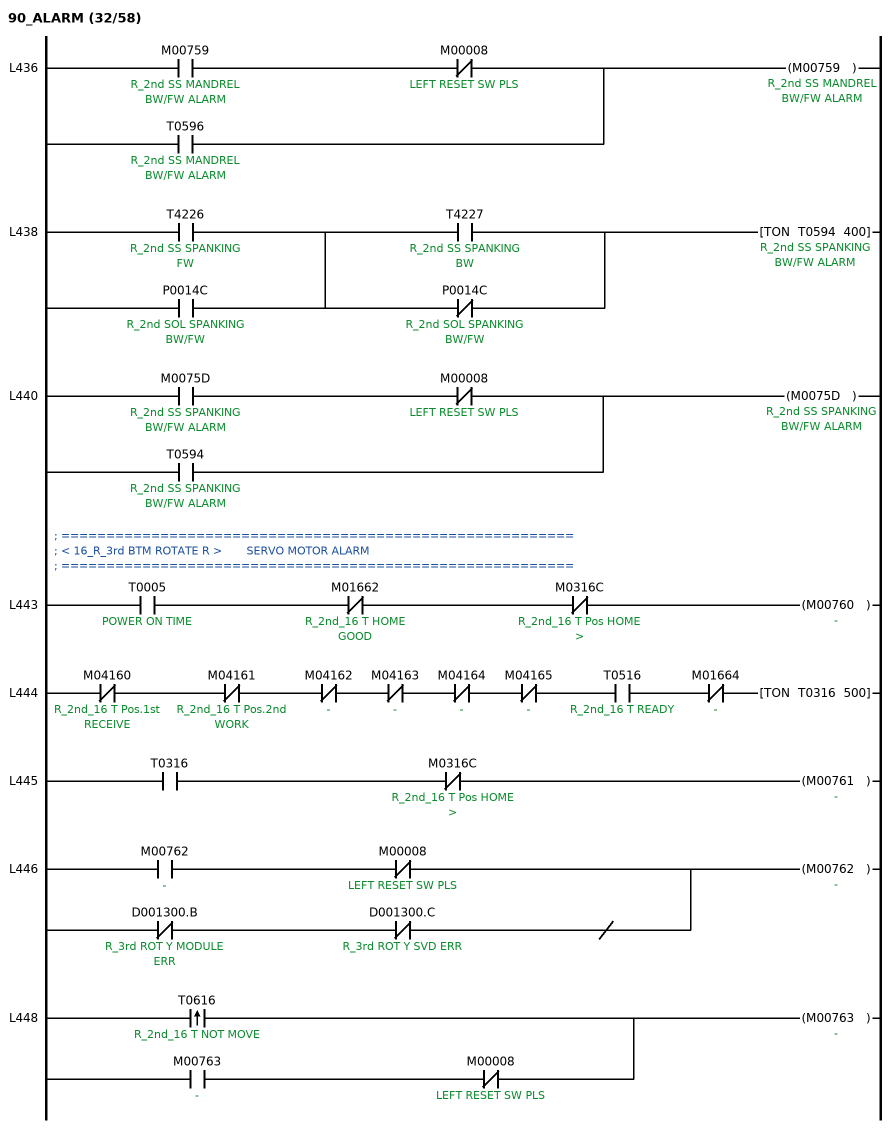
; L436
LOAD      M00759	// R_2nd SS MANDREL BW/FW ALARM
AND NOT   M00008	// LEFT RESET SW PLS
OR        T0596	// R_2nd SS MANDREL BW/FW ALARM
OUT       M00759	// R_2nd SS MANDREL BW/FW ALARM
; L438
LOAD      T4226	// R_2nd SS SPANKING FW
OR        P0014C	// R_2nd SOL SPANKING BW/FW
LOAD      T4227	// R_2nd SS SPANKING BW
OR NOT    P0014C	// R_2nd SOL SPANKING BW/FW
AND LOAD
TON       T0594 400	// R_2nd SS SPANKING BW/FW ALARM
; L440
LOAD      M0075D	// R_2nd SS SPANKING BW/FW ALARM
AND NOT   M00008	// LEFT RESET SW PLS
OR        T0594	// R_2nd SS SPANKING BW/FW ALARM
OUT       M0075D	// R_2nd SS SPANKING BW/FW ALARM
// =========================================================
// 
//        < 16_R_3rd BTM ROTATE R >       SERVO MOTOR ALARM
// 
// =========================================================
; L443
LOAD      T0005	// POWER ON TIME
AND NOT   M01662	// R_2nd_16 T HOME GOOD
AND NOT   M0316C	// R_2nd_16 T Pos HOME >
OUT       M00760	// -
; L444
LOAD NOT  M04160	// R_2nd_16 T Pos.1st RECEIVE
AND NOT   M04161	// R_2nd_16 T Pos.2nd WORK
AND NOT   M04162	// -
AND NOT   M04163	// -
AND NOT   M04164	// -
AND NOT   M04165	// -
AND       T0516	// R_2nd_16 T READY
AND NOT   M01664	// -
TON       T0316 500
; L445
LOAD      T0316
AND NOT   M0316C	// R_2nd_16 T Pos HOME >
OUT       M00761	// -
; L446
LOAD      M00762	// -
AND NOT   M00008	// LEFT RESET SW PLS
LOAD NOT  D001300.B	// R_3rd ROT Y MODULE ERR
AND NOT   D001300.C	// R_3rd ROT Y SVD ERR
NOT
OR LOAD
OUT       M00762	// -
; L448
LOADP     T0616	// R_2nd_16 T NOT MOVE
LOAD      M00763	// -
AND NOT   M00008	// LEFT RESET SW PLS
OR LOAD
OUT       M00763	// -

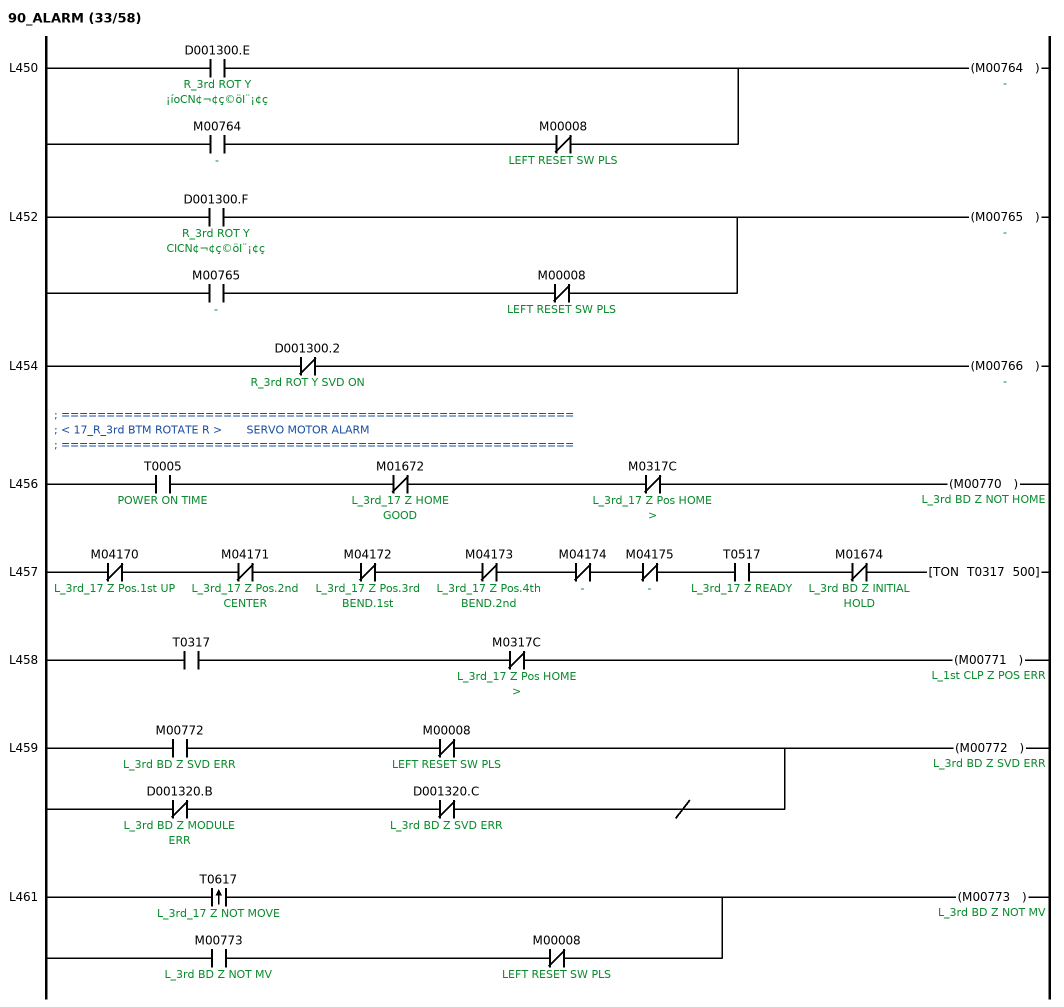
; L450
LOAD      D001300.E	// R_3rd ROT Y ¡íoCN¢¬¢ç©öI¨¡¢ç
LOAD      M00764	// -
AND NOT   M00008	// LEFT RESET SW PLS
OR LOAD
OUT       M00764	// -
; L452
LOAD      D001300.F	// R_3rd ROT Y CICN¢¬¢ç©öI¨¡¢ç
LOAD      M00765	// -
AND NOT   M00008	// LEFT RESET SW PLS
OR LOAD
OUT       M00765	// -
; L454
LOAD NOT  D001300.2	// R_3rd ROT Y SVD ON
OUT       M00766	// -
// =========================================================
// 
//        < 17_R_3rd BTM ROTATE R >       SERVO MOTOR ALARM
// 
// =========================================================
; L456
LOAD      T0005	// POWER ON TIME
AND NOT   M01672	// L_3rd_17 Z HOME GOOD
AND NOT   M0317C	// L_3rd_17 Z Pos HOME >
OUT       M00770	// L_3rd BD Z NOT HOME
; L457
LOAD NOT  M04170	// L_3rd_17 Z Pos.1st UP
AND NOT   M04171	// L_3rd_17 Z Pos.2nd CENTER
AND NOT   M04172	// L_3rd_17 Z Pos.3rd BEND.1st
AND NOT   M04173	// L_3rd_17 Z Pos.4th BEND.2nd
AND NOT   M04174	// -
AND NOT   M04175	// -
AND       T0517	// L_3rd_17 Z READY
AND NOT   M01674	// L_3rd BD Z INITIAL HOLD
TON       T0317 500
; L458
LOAD      T0317
AND NOT   M0317C	// L_3rd_17 Z Pos HOME >
OUT       M00771	// L_1st CLP Z POS ERR
; L459
LOAD      M00772	// L_3rd BD Z SVD ERR
AND NOT   M00008	// LEFT RESET SW PLS
LOAD NOT  D001320.B	// L_3rd BD Z MODULE ERR
AND NOT   D001320.C	// L_3rd BD Z SVD ERR
NOT
OR LOAD
OUT       M00772	// L_3rd BD Z SVD ERR
; L461
LOADP     T0617	// L_3rd_17 Z NOT MOVE
LOAD      M00773	// L_3rd BD Z NOT MV
AND NOT   M00008	// LEFT RESET SW PLS
OR LOAD
OUT       M00773	// L_3rd BD Z NOT MV

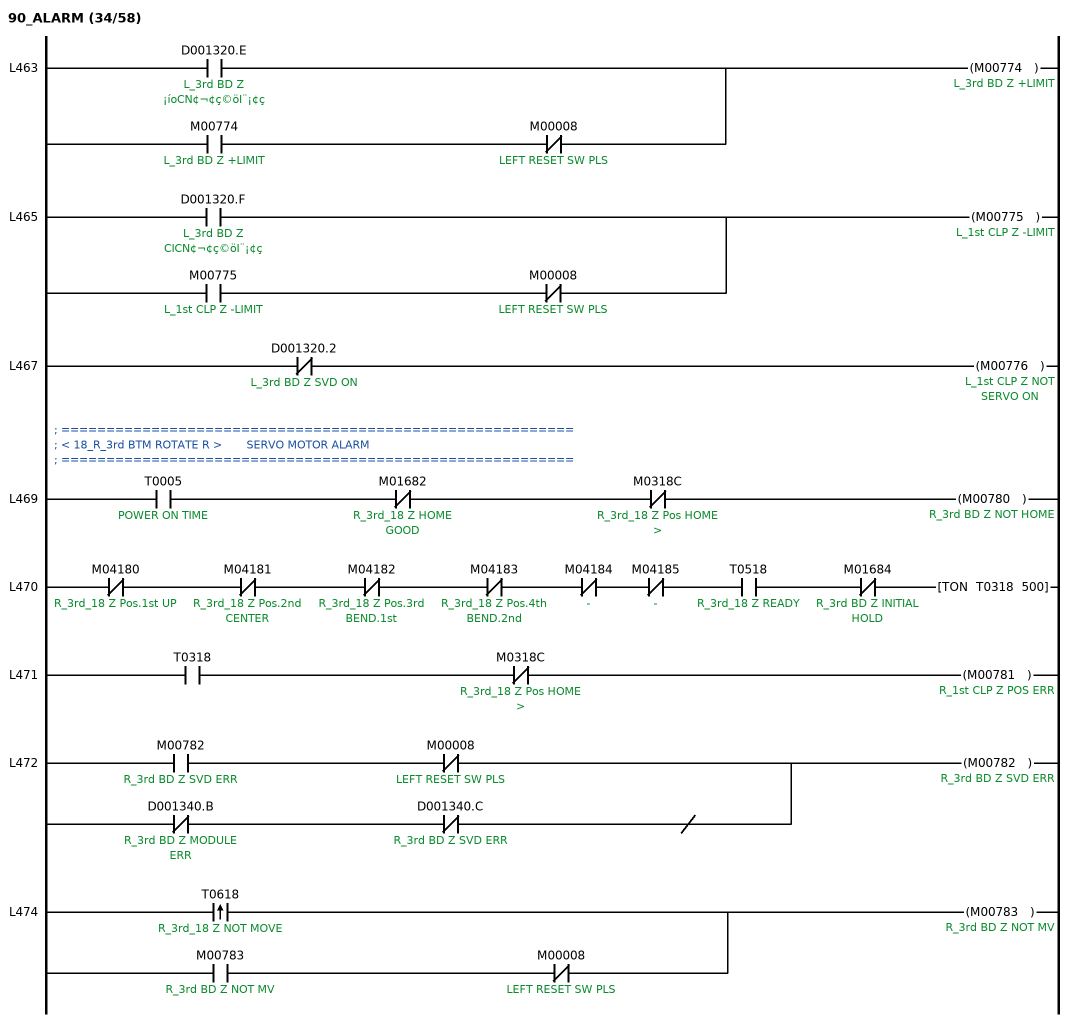
; L463
LOAD      D001320.E	// L_3rd BD Z ¡íoCN¢¬¢ç©öI¨¡¢ç
LOAD      M00774	// L_3rd BD Z +LIMIT
AND NOT   M00008	// LEFT RESET SW PLS
OR LOAD
OUT       M00774	// L_3rd BD Z +LIMIT
; L465
LOAD      D001320.F	// L_3rd BD Z CICN¢¬¢ç©öI¨¡¢ç
LOAD      M00775	// L_1st CLP Z -LIMIT
AND NOT   M00008	// LEFT RESET SW PLS
OR LOAD
OUT       M00775	// L_1st CLP Z -LIMIT
; L467
LOAD NOT  D001320.2	// L_3rd BD Z SVD ON
OUT       M00776	// L_1st CLP Z NOT SERVO ON
// =========================================================
// 
//        < 18_R_3rd BTM ROTATE R >       SERVO MOTOR ALARM
// 
// =========================================================
; L469
LOAD      T0005	// POWER ON TIME
AND NOT   M01682	// R_3rd_18 Z HOME GOOD
AND NOT   M0318C	// R_3rd_18 Z Pos HOME >
OUT       M00780	// R_3rd BD Z NOT HOME
; L470
LOAD NOT  M04180	// R_3rd_18 Z Pos.1st UP
AND NOT   M04181	// R_3rd_18 Z Pos.2nd CENTER
AND NOT   M04182	// R_3rd_18 Z Pos.3rd BEND.1st
AND NOT   M04183	// R_3rd_18 Z Pos.4th BEND.2nd
AND NOT   M04184	// -
AND NOT   M04185	// -
AND       T0518	// R_3rd_18 Z READY
AND NOT   M01684	// R_3rd BD Z INITIAL HOLD
TON       T0318 500
; L471
LOAD      T0318
AND NOT   M0318C	// R_3rd_18 Z Pos HOME >
OUT       M00781	// R_1st CLP Z POS ERR
; L472
LOAD      M00782	// R_3rd BD Z SVD ERR
AND NOT   M00008	// LEFT RESET SW PLS
LOAD NOT  D001340.B	// R_3rd BD Z MODULE ERR
AND NOT   D001340.C	// R_3rd BD Z SVD ERR
NOT
OR LOAD
OUT       M00782	// R_3rd BD Z SVD ERR
; L474
LOADP     T0618	// R_3rd_18 Z NOT MOVE
LOAD      M00783	// R_3rd BD Z NOT MV
AND NOT   M00008	// LEFT RESET SW PLS
OR LOAD
OUT       M00783	// R_3rd BD Z NOT MV

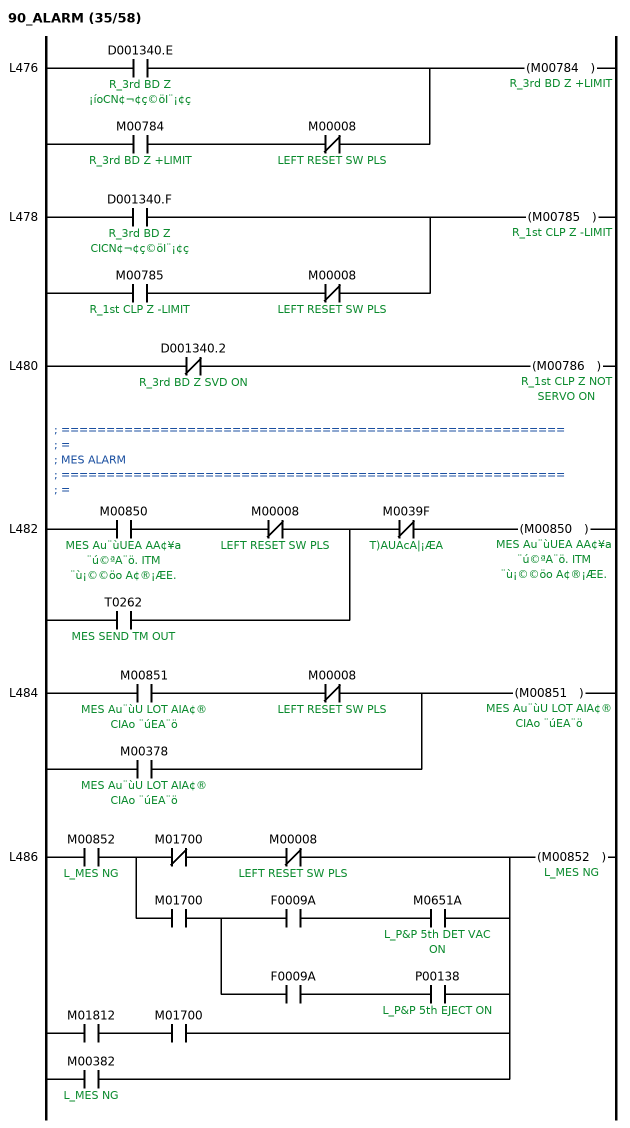
; L476
LOAD      D001340.E	// R_3rd BD Z ¡íoCN¢¬¢ç©öI¨¡¢ç
LOAD      M00784	// R_3rd BD Z +LIMIT
AND NOT   M00008	// LEFT RESET SW PLS
OR LOAD
OUT       M00784	// R_3rd BD Z +LIMIT
; L478
LOAD      D001340.F	// R_3rd BD Z CICN¢¬¢ç©öI¨¡¢ç
LOAD      M00785	// R_1st CLP Z -LIMIT
AND NOT   M00008	// LEFT RESET SW PLS
OR LOAD
OUT       M00785	// R_1st CLP Z -LIMIT
; L480
LOAD NOT  D001340.2	// R_3rd BD Z SVD ON
OUT       M00786	// R_1st CLP Z NOT SERVO ON
// =========================================================
// 
//        MES ALARM
// 
// =========================================================
; L482
LOAD      M00850	// MES Au¨ùUEA AA¢¥a ¨ú©ªA¨ö. ITM ¨ù¡©©öo A¢®¡ÆE.
AND NOT   M00008	// LEFT RESET SW PLS
OR        T0262	// MES SEND TM OUT
AND NOT   M0039F	// T)AUAcA|¡ÆA
OUT       M00850	// MES Au¨ùUEA AA¢¥a ¨ú©ªA¨ö. ITM ¨ù¡©©öo A¢®¡ÆE.
; L484
LOAD      M00851	// MES Au¨ùU LOT AIA¢® CIAo ¨úEA¨ö
AND NOT   M00008	// LEFT RESET SW PLS
OR        M00378	// MES Au¨ùU LOT AIA¢® CIAo ¨úEA¨ö
OUT       M00851	// MES Au¨ùU LOT AIA¢® CIAo ¨úEA¨ö
; L486
LOAD      M00852	// L_MES NG
LOAD NOT  M01700
AND NOT   M00008	// LEFT RESET SW PLS
LOAD      M01700
LOAD      F0009A
AND       M0651A	// L_P&P 5th DET VAC ON
LOAD      F0009A
AND       P00138	// L_P&P 5th EJECT ON
OR LOAD
AND LOAD
OR LOAD
AND LOAD
LOAD      M01812
AND       M01700
OR LOAD
OR        M00382	// L_MES NG
OUT       M00852	// L_MES NG

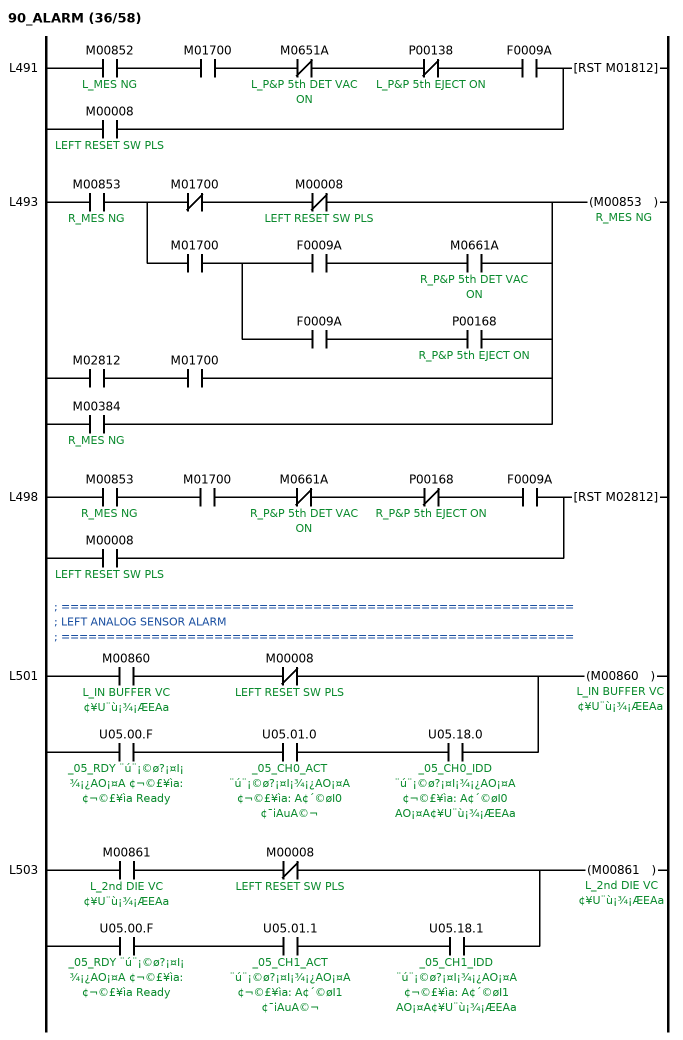
; L491
LOAD      M00852	// L_MES NG
AND       M01700
AND NOT   M0651A	// L_P&P 5th DET VAC ON
AND NOT   P00138	// L_P&P 5th EJECT ON
AND       F0009A
OR        M00008	// LEFT RESET SW PLS
RST       M01812
; L493
LOAD      M00853	// R_MES NG
LOAD NOT  M01700
AND NOT   M00008	// LEFT RESET SW PLS
LOAD      M01700
LOAD      F0009A
AND       M0661A	// R_P&P 5th DET VAC ON
LOAD      F0009A
AND       P00168	// R_P&P 5th EJECT ON
OR LOAD
AND LOAD
OR LOAD
AND LOAD
LOAD      M02812
AND       M01700
OR LOAD
OR        M00384	// R_MES NG
OUT       M00853	// R_MES NG
; L498
LOAD      M00853	// R_MES NG
AND       M01700
AND NOT   M0661A	// R_P&P 5th DET VAC ON
AND NOT   P00168	// R_P&P 5th EJECT ON
AND       F0009A
OR        M00008	// LEFT RESET SW PLS
RST       M02812
// =========================================================
// 
//        LEFT ANALOG SENSOR ALARM
// 
// =========================================================
; L501
LOAD      M00860	// L_IN BUFFER VC ¢¥U¨ù¡¾¡ÆEAa
AND NOT   M00008	// LEFT RESET SW PLS
LOAD      U05.00.F	// _05_RDY ¨ú¨¡©ø?¡¤I¡¾¡¿AO¡¤A ¢¬©£¥ìa: ¢¬©£¥ìa Ready
AND       U05.01.0	// _05_CH0_ACT ¨ú¨¡©ø?¡¤I¡¾¡¿AO¡¤A ¢¬©£¥ìa: A¢´©øI0 ¢¯iAuA©¬
AND       U05.18.0	// _05_CH0_IDD ¨ú¨¡©ø?¡¤I¡¾¡¿AO¡¤A ¢¬©£¥ìa: A¢´©øI0 AO¡¤A¢¥U¨ù¡¾¡ÆEAa
OR LOAD
OUT       M00860	// L_IN BUFFER VC ¢¥U¨ù¡¾¡ÆEAa
; L503
LOAD      M00861	// L_2nd DIE VC ¢¥U¨ù¡¾¡ÆEAa
AND NOT   M00008	// LEFT RESET SW PLS
LOAD      U05.00.F	// _05_RDY ¨ú¨¡©ø?¡¤I¡¾¡¿AO¡¤A ¢¬©£¥ìa: ¢¬©£¥ìa Ready
AND       U05.01.1	// _05_CH1_ACT ¨ú¨¡©ø?¡¤I¡¾¡¿AO¡¤A ¢¬©£¥ìa: A¢´©øI1 ¢¯iAuA©¬
AND       U05.18.1	// _05_CH1_IDD ¨ú¨¡©ø?¡¤I¡¾¡¿AO¡¤A ¢¬©£¥ìa: A¢´©øI1 AO¡¤A¢¥U¨ù¡¾¡ÆEAa
OR LOAD
OUT       M00861	// L_2nd DIE VC ¢¥U¨ù¡¾¡ÆEAa

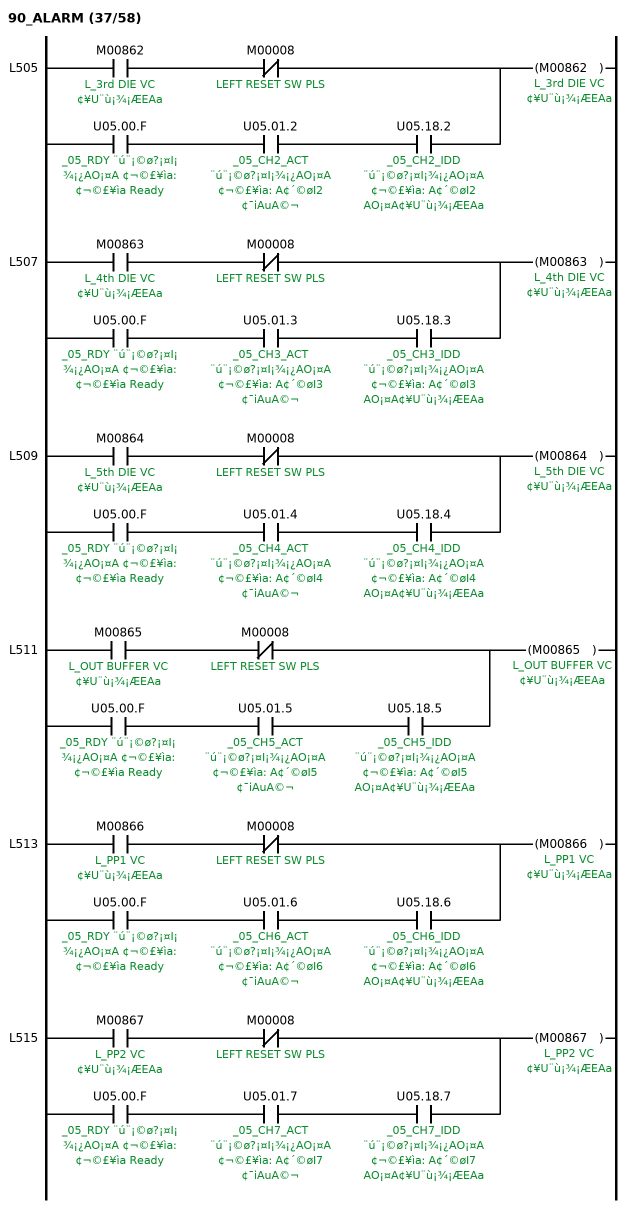
; L505
LOAD      M00862	// L_3rd DIE VC ¢¥U¨ù¡¾¡ÆEAa
AND NOT   M00008	// LEFT RESET SW PLS
LOAD      U05.00.F	// _05_RDY ¨ú¨¡©ø?¡¤I¡¾¡¿AO¡¤A ¢¬©£¥ìa: ¢¬©£¥ìa Ready
AND       U05.01.2	// _05_CH2_ACT ¨ú¨¡©ø?¡¤I¡¾¡¿AO¡¤A ¢¬©£¥ìa: A¢´©øI2 ¢¯iAuA©¬
AND       U05.18.2	// _05_CH2_IDD ¨ú¨¡©ø?¡¤I¡¾¡¿AO¡¤A ¢¬©£¥ìa: A¢´©øI2 AO¡¤A¢¥U¨ù¡¾¡ÆEAa
OR LOAD
OUT       M00862	// L_3rd DIE VC ¢¥U¨ù¡¾¡ÆEAa
; L507
LOAD      M00863	// L_4th DIE VC ¢¥U¨ù¡¾¡ÆEAa
AND NOT   M00008	// LEFT RESET SW PLS
LOAD      U05.00.F	// _05_RDY ¨ú¨¡©ø?¡¤I¡¾¡¿AO¡¤A ¢¬©£¥ìa: ¢¬©£¥ìa Ready
AND       U05.01.3	// _05_CH3_ACT ¨ú¨¡©ø?¡¤I¡¾¡¿AO¡¤A ¢¬©£¥ìa: A¢´©øI3 ¢¯iAuA©¬
AND       U05.18.3	// _05_CH3_IDD ¨ú¨¡©ø?¡¤I¡¾¡¿AO¡¤A ¢¬©£¥ìa: A¢´©øI3 AO¡¤A¢¥U¨ù¡¾¡ÆEAa
OR LOAD
OUT       M00863	// L_4th DIE VC ¢¥U¨ù¡¾¡ÆEAa
; L509
LOAD      M00864	// L_5th DIE VC ¢¥U¨ù¡¾¡ÆEAa
AND NOT   M00008	// LEFT RESET SW PLS
LOAD      U05.00.F	// _05_RDY ¨ú¨¡©ø?¡¤I¡¾¡¿AO¡¤A ¢¬©£¥ìa: ¢¬©£¥ìa Ready
AND       U05.01.4	// _05_CH4_ACT ¨ú¨¡©ø?¡¤I¡¾¡¿AO¡¤A ¢¬©£¥ìa: A¢´©øI4 ¢¯iAuA©¬
AND       U05.18.4	// _05_CH4_IDD ¨ú¨¡©ø?¡¤I¡¾¡¿AO¡¤A ¢¬©£¥ìa: A¢´©øI4 AO¡¤A¢¥U¨ù¡¾¡ÆEAa
OR LOAD
OUT       M00864	// L_5th DIE VC ¢¥U¨ù¡¾¡ÆEAa
; L511
LOAD      M00865	// L_OUT BUFFER VC ¢¥U¨ù¡¾¡ÆEAa
AND NOT   M00008	// LEFT RESET SW PLS
LOAD      U05.00.F	// _05_RDY ¨ú¨¡©ø?¡¤I¡¾¡¿AO¡¤A ¢¬©£¥ìa: ¢¬©£¥ìa Ready
AND       U05.01.5	// _05_CH5_ACT ¨ú¨¡©ø?¡¤I¡¾¡¿AO¡¤A ¢¬©£¥ìa: A¢´©øI5 ¢¯iAuA©¬
AND       U05.18.5	// _05_CH5_IDD ¨ú¨¡©ø?¡¤I¡¾¡¿AO¡¤A ¢¬©£¥ìa: A¢´©øI5 AO¡¤A¢¥U¨ù¡¾¡ÆEAa
OR LOAD
OUT       M00865	// L_OUT BUFFER VC ¢¥U¨ù¡¾¡ÆEAa
; L513
LOAD      M00866	// L_PP1 VC ¢¥U¨ù¡¾¡ÆEAa
AND NOT   M00008	// LEFT RESET SW PLS
LOAD      U05.00.F	// _05_RDY ¨ú¨¡©ø?¡¤I¡¾¡¿AO¡¤A ¢¬©£¥ìa: ¢¬©£¥ìa Ready
AND       U05.01.6	// _05_CH6_ACT ¨ú¨¡©ø?¡¤I¡¾¡¿AO¡¤A ¢¬©£¥ìa: A¢´©øI6 ¢¯iAuA©¬
AND       U05.18.6	// _05_CH6_IDD ¨ú¨¡©ø?¡¤I¡¾¡¿AO¡¤A ¢¬©£¥ìa: A¢´©øI6 AO¡¤A¢¥U¨ù¡¾¡ÆEAa
OR LOAD
OUT       M00866	// L_PP1 VC ¢¥U¨ù¡¾¡ÆEAa
; L515
LOAD      M00867	// L_PP2 VC ¢¥U¨ù¡¾¡ÆEAa
AND NOT   M00008	// LEFT RESET SW PLS
LOAD      U05.00.F	// _05_RDY ¨ú¨¡©ø?¡¤I¡¾¡¿AO¡¤A ¢¬©£¥ìa: ¢¬©£¥ìa Ready
AND       U05.01.7	// _05_CH7_ACT ¨ú¨¡©ø?¡¤I¡¾¡¿AO¡¤A ¢¬©£¥ìa: A¢´©øI7 ¢¯iAuA©¬
AND       U05.18.7	// _05_CH7_IDD ¨ú¨¡©ø?¡¤I¡¾¡¿AO¡¤A ¢¬©£¥ìa: A¢´©øI7 AO¡¤A¢¥U¨ù¡¾¡ÆEAa
OR LOAD
OUT       M00867	// L_PP2 VC ¢¥U¨ù¡¾¡ÆEAa

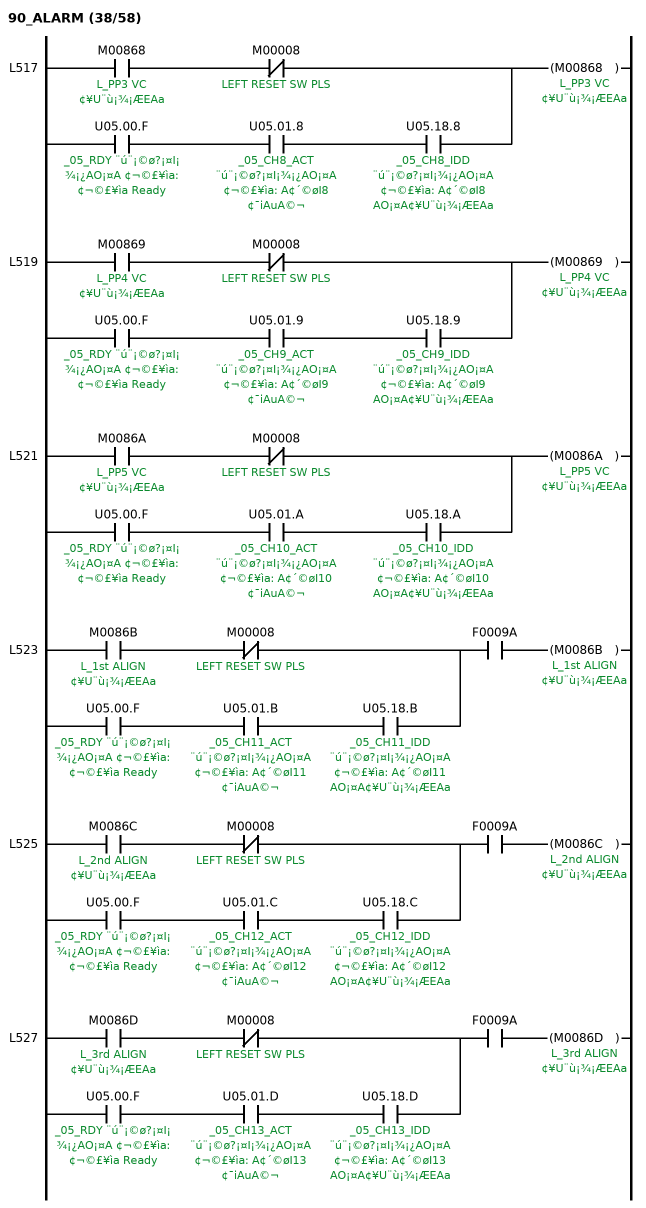
; L517
LOAD      M00868	// L_PP3 VC ¢¥U¨ù¡¾¡ÆEAa
AND NOT   M00008	// LEFT RESET SW PLS
LOAD      U05.00.F	// _05_RDY ¨ú¨¡©ø?¡¤I¡¾¡¿AO¡¤A ¢¬©£¥ìa: ¢¬©£¥ìa Ready
AND       U05.01.8	// _05_CH8_ACT ¨ú¨¡©ø?¡¤I¡¾¡¿AO¡¤A ¢¬©£¥ìa: A¢´©øI8 ¢¯iAuA©¬
AND       U05.18.8	// _05_CH8_IDD ¨ú¨¡©ø?¡¤I¡¾¡¿AO¡¤A ¢¬©£¥ìa: A¢´©øI8 AO¡¤A¢¥U¨ù¡¾¡ÆEAa
OR LOAD
OUT       M00868	// L_PP3 VC ¢¥U¨ù¡¾¡ÆEAa
; L519
LOAD      M00869	// L_PP4 VC ¢¥U¨ù¡¾¡ÆEAa
AND NOT   M00008	// LEFT RESET SW PLS
LOAD      U05.00.F	// _05_RDY ¨ú¨¡©ø?¡¤I¡¾¡¿AO¡¤A ¢¬©£¥ìa: ¢¬©£¥ìa Ready
AND       U05.01.9	// _05_CH9_ACT ¨ú¨¡©ø?¡¤I¡¾¡¿AO¡¤A ¢¬©£¥ìa: A¢´©øI9 ¢¯iAuA©¬
AND       U05.18.9	// _05_CH9_IDD ¨ú¨¡©ø?¡¤I¡¾¡¿AO¡¤A ¢¬©£¥ìa: A¢´©øI9 AO¡¤A¢¥U¨ù¡¾¡ÆEAa
OR LOAD
OUT       M00869	// L_PP4 VC ¢¥U¨ù¡¾¡ÆEAa
; L521
LOAD      M0086A	// L_PP5 VC ¢¥U¨ù¡¾¡ÆEAa
AND NOT   M00008	// LEFT RESET SW PLS
LOAD      U05.00.F	// _05_RDY ¨ú¨¡©ø?¡¤I¡¾¡¿AO¡¤A ¢¬©£¥ìa: ¢¬©£¥ìa Ready
AND       U05.01.A	// _05_CH10_ACT ¨ú¨¡©ø?¡¤I¡¾¡¿AO¡¤A ¢¬©£¥ìa: A¢´©øI10 ¢¯iAuA©¬
AND       U05.18.A	// _05_CH10_IDD ¨ú¨¡©ø?¡¤I¡¾¡¿AO¡¤A ¢¬©£¥ìa: A¢´©øI10 AO¡¤A¢¥U¨ù¡¾¡ÆEAa
OR LOAD
OUT       M0086A	// L_PP5 VC ¢¥U¨ù¡¾¡ÆEAa
; L523
LOAD      M0086B	// L_1st ALIGN ¢¥U¨ù¡¾¡ÆEAa
AND NOT   M00008	// LEFT RESET SW PLS
LOAD      U05.00.F	// _05_RDY ¨ú¨¡©ø?¡¤I¡¾¡¿AO¡¤A ¢¬©£¥ìa: ¢¬©£¥ìa Ready
AND       U05.01.B	// _05_CH11_ACT ¨ú¨¡©ø?¡¤I¡¾¡¿AO¡¤A ¢¬©£¥ìa: A¢´©øI11 ¢¯iAuA©¬
AND       U05.18.B	// _05_CH11_IDD ¨ú¨¡©ø?¡¤I¡¾¡¿AO¡¤A ¢¬©£¥ìa: A¢´©øI11 AO¡¤A¢¥U¨ù¡¾¡ÆEAa
OR LOAD
AND       F0009A
OUT       M0086B	// L_1st ALIGN ¢¥U¨ù¡¾¡ÆEAa
; L525
LOAD      M0086C	// L_2nd ALIGN ¢¥U¨ù¡¾¡ÆEAa
AND NOT   M00008	// LEFT RESET SW PLS
LOAD      U05.00.F	// _05_RDY ¨ú¨¡©ø?¡¤I¡¾¡¿AO¡¤A ¢¬©£¥ìa: ¢¬©£¥ìa Ready
AND       U05.01.C	// _05_CH12_ACT ¨ú¨¡©ø?¡¤I¡¾¡¿AO¡¤A ¢¬©£¥ìa: A¢´©øI12 ¢¯iAuA©¬
AND       U05.18.C	// _05_CH12_IDD ¨ú¨¡©ø?¡¤I¡¾¡¿AO¡¤A ¢¬©£¥ìa: A¢´©øI12 AO¡¤A¢¥U¨ù¡¾¡ÆEAa
OR LOAD
AND       F0009A
OUT       M0086C	// L_2nd ALIGN ¢¥U¨ù¡¾¡ÆEAa
; L527
LOAD      M0086D	// L_3rd ALIGN ¢¥U¨ù¡¾¡ÆEAa
AND NOT   M00008	// LEFT RESET SW PLS
LOAD      U05.00.F	// _05_RDY ¨ú¨¡©ø?¡¤I¡¾¡¿AO¡¤A ¢¬©£¥ìa: ¢¬©£¥ìa Ready
AND       U05.01.D	// _05_CH13_ACT ¨ú¨¡©ø?¡¤I¡¾¡¿AO¡¤A ¢¬©£¥ìa: A¢´©øI13 ¢¯iAuA©¬
AND       U05.18.D	// _05_CH13_IDD ¨ú¨¡©ø?¡¤I¡¾¡¿AO¡¤A ¢¬©£¥ìa: A¢´©øI13 AO¡¤A¢¥U¨ù¡¾¡ÆEAa
OR LOAD
AND       F0009A
OUT       M0086D	// L_3rd ALIGN ¢¥U¨ù¡¾¡ÆEAa

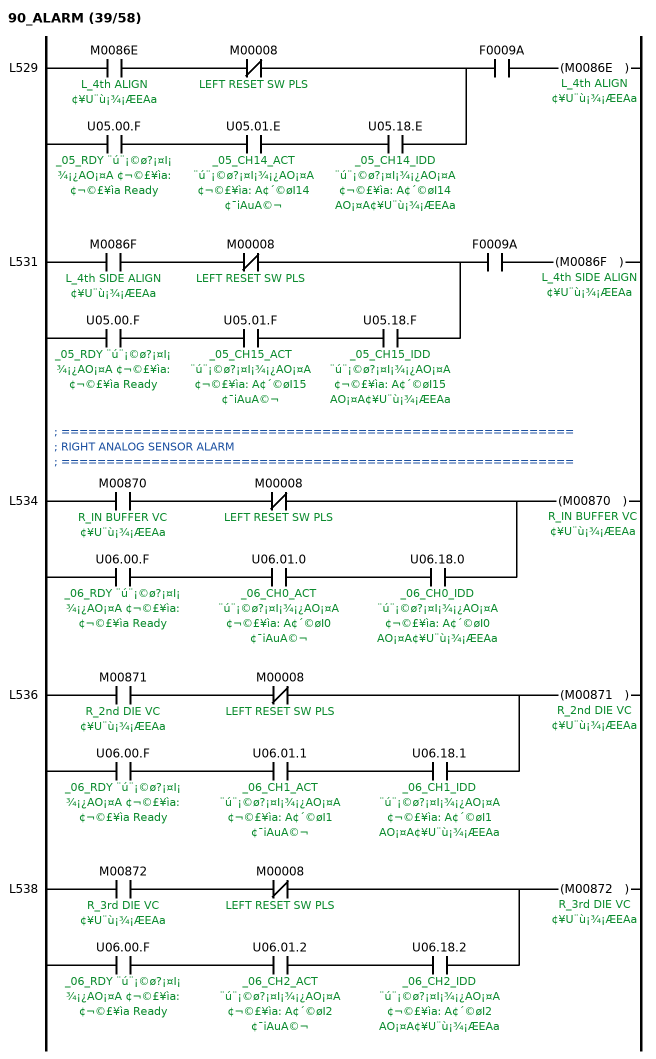
; L529
LOAD      M0086E	// L_4th ALIGN ¢¥U¨ù¡¾¡ÆEAa
AND NOT   M00008	// LEFT RESET SW PLS
LOAD      U05.00.F	// _05_RDY ¨ú¨¡©ø?¡¤I¡¾¡¿AO¡¤A ¢¬©£¥ìa: ¢¬©£¥ìa Ready
AND       U05.01.E	// _05_CH14_ACT ¨ú¨¡©ø?¡¤I¡¾¡¿AO¡¤A ¢¬©£¥ìa: A¢´©øI14 ¢¯iAuA©¬
AND       U05.18.E	// _05_CH14_IDD ¨ú¨¡©ø?¡¤I¡¾¡¿AO¡¤A ¢¬©£¥ìa: A¢´©øI14 AO¡¤A¢¥U¨ù¡¾¡ÆEAa
OR LOAD
AND       F0009A
OUT       M0086E	// L_4th ALIGN ¢¥U¨ù¡¾¡ÆEAa
; L531
LOAD      M0086F	// L_4th SIDE ALIGN ¢¥U¨ù¡¾¡ÆEAa
AND NOT   M00008	// LEFT RESET SW PLS
LOAD      U05.00.F	// _05_RDY ¨ú¨¡©ø?¡¤I¡¾¡¿AO¡¤A ¢¬©£¥ìa: ¢¬©£¥ìa Ready
AND       U05.01.F	// _05_CH15_ACT ¨ú¨¡©ø?¡¤I¡¾¡¿AO¡¤A ¢¬©£¥ìa: A¢´©øI15 ¢¯iAuA©¬
AND       U05.18.F	// _05_CH15_IDD ¨ú¨¡©ø?¡¤I¡¾¡¿AO¡¤A ¢¬©£¥ìa: A¢´©øI15 AO¡¤A¢¥U¨ù¡¾¡ÆEAa
OR LOAD
AND       F0009A
OUT       M0086F	// L_4th SIDE ALIGN ¢¥U¨ù¡¾¡ÆEAa
// =========================================================
// 
//        RIGHT ANALOG SENSOR ALARM
// 
// =========================================================
; L534
LOAD      M00870	// R_IN BUFFER VC ¢¥U¨ù¡¾¡ÆEAa
AND NOT   M00008	// LEFT RESET SW PLS
LOAD      U06.00.F	// _06_RDY ¨ú¨¡©ø?¡¤I¡¾¡¿AO¡¤A ¢¬©£¥ìa: ¢¬©£¥ìa Ready
AND       U06.01.0	// _06_CH0_ACT ¨ú¨¡©ø?¡¤I¡¾¡¿AO¡¤A ¢¬©£¥ìa: A¢´©øI0 ¢¯iAuA©¬
AND       U06.18.0	// _06_CH0_IDD ¨ú¨¡©ø?¡¤I¡¾¡¿AO¡¤A ¢¬©£¥ìa: A¢´©øI0 AO¡¤A¢¥U¨ù¡¾¡ÆEAa
OR LOAD
OUT       M00870	// R_IN BUFFER VC ¢¥U¨ù¡¾¡ÆEAa
; L536
LOAD      M00871	// R_2nd DIE VC ¢¥U¨ù¡¾¡ÆEAa
AND NOT   M00008	// LEFT RESET SW PLS
LOAD      U06.00.F	// _06_RDY ¨ú¨¡©ø?¡¤I¡¾¡¿AO¡¤A ¢¬©£¥ìa: ¢¬©£¥ìa Ready
AND       U06.01.1	// _06_CH1_ACT ¨ú¨¡©ø?¡¤I¡¾¡¿AO¡¤A ¢¬©£¥ìa: A¢´©øI1 ¢¯iAuA©¬
AND       U06.18.1	// _06_CH1_IDD ¨ú¨¡©ø?¡¤I¡¾¡¿AO¡¤A ¢¬©£¥ìa: A¢´©øI1 AO¡¤A¢¥U¨ù¡¾¡ÆEAa
OR LOAD
OUT       M00871	// R_2nd DIE VC ¢¥U¨ù¡¾¡ÆEAa
; L538
LOAD      M00872	// R_3rd DIE VC ¢¥U¨ù¡¾¡ÆEAa
AND NOT   M00008	// LEFT RESET SW PLS
LOAD      U06.00.F	// _06_RDY ¨ú¨¡©ø?¡¤I¡¾¡¿AO¡¤A ¢¬©£¥ìa: ¢¬©£¥ìa Ready
AND       U06.01.2	// _06_CH2_ACT ¨ú¨¡©ø?¡¤I¡¾¡¿AO¡¤A ¢¬©£¥ìa: A¢´©øI2 ¢¯iAuA©¬
AND       U06.18.2	// _06_CH2_IDD ¨ú¨¡©ø?¡¤I¡¾¡¿AO¡¤A ¢¬©£¥ìa: A¢´©øI2 AO¡¤A¢¥U¨ù¡¾¡ÆEAa
OR LOAD
OUT       M00872	// R_3rd DIE VC ¢¥U¨ù¡¾¡ÆEAa

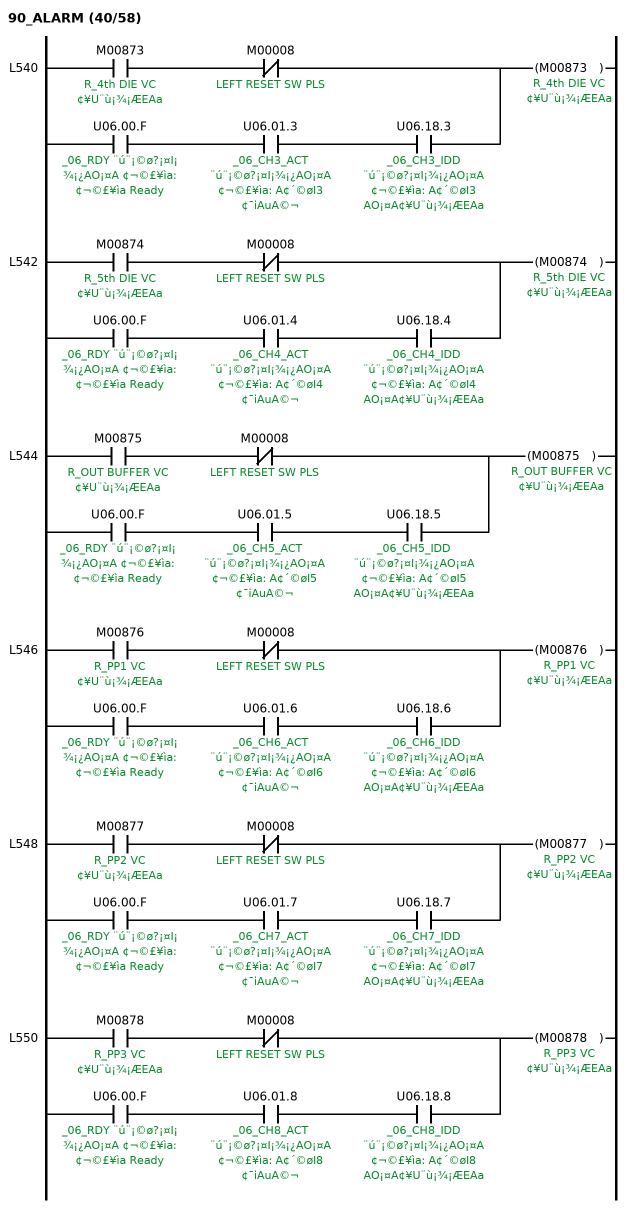
; L540
LOAD      M00873	// R_4th DIE VC ¢¥U¨ù¡¾¡ÆEAa
AND NOT   M00008	// LEFT RESET SW PLS
LOAD      U06.00.F	// _06_RDY ¨ú¨¡©ø?¡¤I¡¾¡¿AO¡¤A ¢¬©£¥ìa: ¢¬©£¥ìa Ready
AND       U06.01.3	// _06_CH3_ACT ¨ú¨¡©ø?¡¤I¡¾¡¿AO¡¤A ¢¬©£¥ìa: A¢´©øI3 ¢¯iAuA©¬
AND       U06.18.3	// _06_CH3_IDD ¨ú¨¡©ø?¡¤I¡¾¡¿AO¡¤A ¢¬©£¥ìa: A¢´©øI3 AO¡¤A¢¥U¨ù¡¾¡ÆEAa
OR LOAD
OUT       M00873	// R_4th DIE VC ¢¥U¨ù¡¾¡ÆEAa
; L542
LOAD      M00874	// R_5th DIE VC ¢¥U¨ù¡¾¡ÆEAa
AND NOT   M00008	// LEFT RESET SW PLS
LOAD      U06.00.F	// _06_RDY ¨ú¨¡©ø?¡¤I¡¾¡¿AO¡¤A ¢¬©£¥ìa: ¢¬©£¥ìa Ready
AND       U06.01.4	// _06_CH4_ACT ¨ú¨¡©ø?¡¤I¡¾¡¿AO¡¤A ¢¬©£¥ìa: A¢´©øI4 ¢¯iAuA©¬
AND       U06.18.4	// _06_CH4_IDD ¨ú¨¡©ø?¡¤I¡¾¡¿AO¡¤A ¢¬©£¥ìa: A¢´©øI4 AO¡¤A¢¥U¨ù¡¾¡ÆEAa
OR LOAD
OUT       M00874	// R_5th DIE VC ¢¥U¨ù¡¾¡ÆEAa
; L544
LOAD      M00875	// R_OUT BUFFER VC ¢¥U¨ù¡¾¡ÆEAa
AND NOT   M00008	// LEFT RESET SW PLS
LOAD      U06.00.F	// _06_RDY ¨ú¨¡©ø?¡¤I¡¾¡¿AO¡¤A ¢¬©£¥ìa: ¢¬©£¥ìa Ready
AND       U06.01.5	// _06_CH5_ACT ¨ú¨¡©ø?¡¤I¡¾¡¿AO¡¤A ¢¬©£¥ìa: A¢´©øI5 ¢¯iAuA©¬
AND       U06.18.5	// _06_CH5_IDD ¨ú¨¡©ø?¡¤I¡¾¡¿AO¡¤A ¢¬©£¥ìa: A¢´©øI5 AO¡¤A¢¥U¨ù¡¾¡ÆEAa
OR LOAD
OUT       M00875	// R_OUT BUFFER VC ¢¥U¨ù¡¾¡ÆEAa
; L546
LOAD      M00876	// R_PP1 VC ¢¥U¨ù¡¾¡ÆEAa
AND NOT   M00008	// LEFT RESET SW PLS
LOAD      U06.00.F	// _06_RDY ¨ú¨¡©ø?¡¤I¡¾¡¿AO¡¤A ¢¬©£¥ìa: ¢¬©£¥ìa Ready
AND       U06.01.6	// _06_CH6_ACT ¨ú¨¡©ø?¡¤I¡¾¡¿AO¡¤A ¢¬©£¥ìa: A¢´©øI6 ¢¯iAuA©¬
AND       U06.18.6	// _06_CH6_IDD ¨ú¨¡©ø?¡¤I¡¾¡¿AO¡¤A ¢¬©£¥ìa: A¢´©øI6 AO¡¤A¢¥U¨ù¡¾¡ÆEAa
OR LOAD
OUT       M00876	// R_PP1 VC ¢¥U¨ù¡¾¡ÆEAa
; L548
LOAD      M00877	// R_PP2 VC ¢¥U¨ù¡¾¡ÆEAa
AND NOT   M00008	// LEFT RESET SW PLS
LOAD      U06.00.F	// _06_RDY ¨ú¨¡©ø?¡¤I¡¾¡¿AO¡¤A ¢¬©£¥ìa: ¢¬©£¥ìa Ready
AND       U06.01.7	// _06_CH7_ACT ¨ú¨¡©ø?¡¤I¡¾¡¿AO¡¤A ¢¬©£¥ìa: A¢´©øI7 ¢¯iAuA©¬
AND       U06.18.7	// _06_CH7_IDD ¨ú¨¡©ø?¡¤I¡¾¡¿AO¡¤A ¢¬©£¥ìa: A¢´©øI7 AO¡¤A¢¥U¨ù¡¾¡ÆEAa
OR LOAD
OUT       M00877	// R_PP2 VC ¢¥U¨ù¡¾¡ÆEAa
; L550
LOAD      M00878	// R_PP3 VC ¢¥U¨ù¡¾¡ÆEAa
AND NOT   M00008	// LEFT RESET SW PLS
LOAD      U06.00.F	// _06_RDY ¨ú¨¡©ø?¡¤I¡¾¡¿AO¡¤A ¢¬©£¥ìa: ¢¬©£¥ìa Ready
AND       U06.01.8	// _06_CH8_ACT ¨ú¨¡©ø?¡¤I¡¾¡¿AO¡¤A ¢¬©£¥ìa: A¢´©øI8 ¢¯iAuA©¬
AND       U06.18.8	// _06_CH8_IDD ¨ú¨¡©ø?¡¤I¡¾¡¿AO¡¤A ¢¬©£¥ìa: A¢´©øI8 AO¡¤A¢¥U¨ù¡¾¡ÆEAa
OR LOAD
OUT       M00878	// R_PP3 VC ¢¥U¨ù¡¾¡ÆEAa

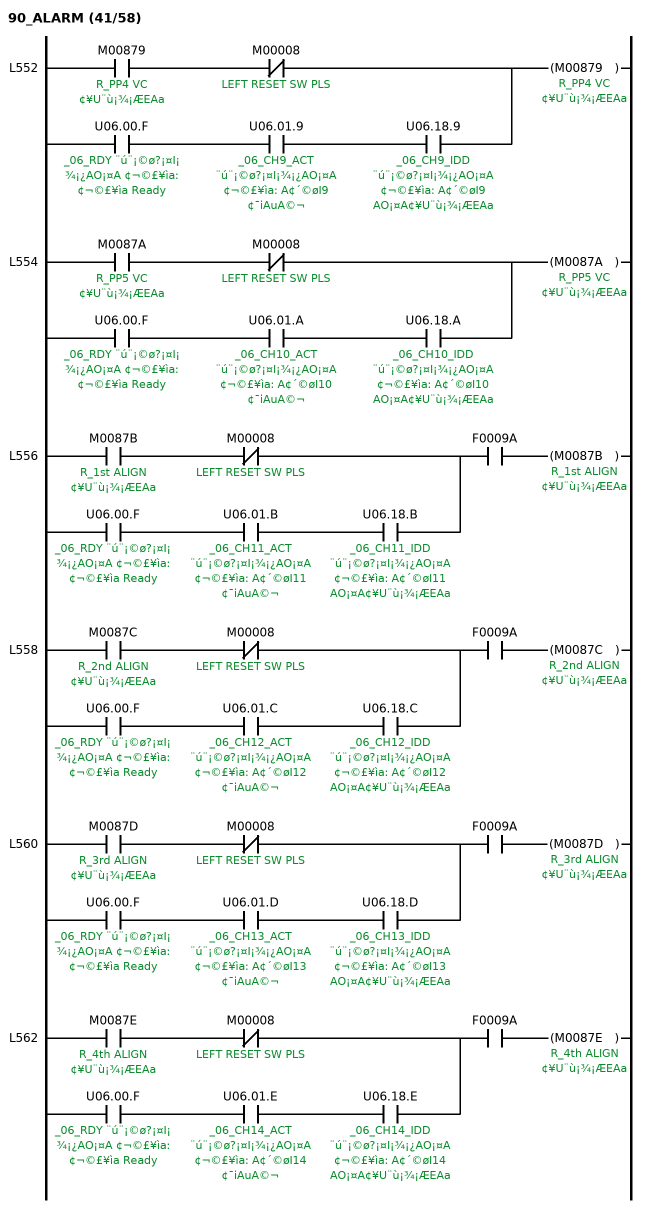
; L552
LOAD      M00879	// R_PP4 VC ¢¥U¨ù¡¾¡ÆEAa
AND NOT   M00008	// LEFT RESET SW PLS
LOAD      U06.00.F	// _06_RDY ¨ú¨¡©ø?¡¤I¡¾¡¿AO¡¤A ¢¬©£¥ìa: ¢¬©£¥ìa Ready
AND       U06.01.9	// _06_CH9_ACT ¨ú¨¡©ø?¡¤I¡¾¡¿AO¡¤A ¢¬©£¥ìa: A¢´©øI9 ¢¯iAuA©¬
AND       U06.18.9	// _06_CH9_IDD ¨ú¨¡©ø?¡¤I¡¾¡¿AO¡¤A ¢¬©£¥ìa: A¢´©øI9 AO¡¤A¢¥U¨ù¡¾¡ÆEAa
OR LOAD
OUT       M00879	// R_PP4 VC ¢¥U¨ù¡¾¡ÆEAa
; L554
LOAD      M0087A	// R_PP5 VC ¢¥U¨ù¡¾¡ÆEAa
AND NOT   M00008	// LEFT RESET SW PLS
LOAD      U06.00.F	// _06_RDY ¨ú¨¡©ø?¡¤I¡¾¡¿AO¡¤A ¢¬©£¥ìa: ¢¬©£¥ìa Ready
AND       U06.01.A	// _06_CH10_ACT ¨ú¨¡©ø?¡¤I¡¾¡¿AO¡¤A ¢¬©£¥ìa: A¢´©øI10 ¢¯iAuA©¬
AND       U06.18.A	// _06_CH10_IDD ¨ú¨¡©ø?¡¤I¡¾¡¿AO¡¤A ¢¬©£¥ìa: A¢´©øI10 AO¡¤A¢¥U¨ù¡¾¡ÆEAa
OR LOAD
OUT       M0087A	// R_PP5 VC ¢¥U¨ù¡¾¡ÆEAa
; L556
LOAD      M0087B	// R_1st ALIGN ¢¥U¨ù¡¾¡ÆEAa
AND NOT   M00008	// LEFT RESET SW PLS
LOAD      U06.00.F	// _06_RDY ¨ú¨¡©ø?¡¤I¡¾¡¿AO¡¤A ¢¬©£¥ìa: ¢¬©£¥ìa Ready
AND       U06.01.B	// _06_CH11_ACT ¨ú¨¡©ø?¡¤I¡¾¡¿AO¡¤A ¢¬©£¥ìa: A¢´©øI11 ¢¯iAuA©¬
AND       U06.18.B	// _06_CH11_IDD ¨ú¨¡©ø?¡¤I¡¾¡¿AO¡¤A ¢¬©£¥ìa: A¢´©øI11 AO¡¤A¢¥U¨ù¡¾¡ÆEAa
OR LOAD
AND       F0009A
OUT       M0087B	// R_1st ALIGN ¢¥U¨ù¡¾¡ÆEAa
; L558
LOAD      M0087C	// R_2nd ALIGN ¢¥U¨ù¡¾¡ÆEAa
AND NOT   M00008	// LEFT RESET SW PLS
LOAD      U06.00.F	// _06_RDY ¨ú¨¡©ø?¡¤I¡¾¡¿AO¡¤A ¢¬©£¥ìa: ¢¬©£¥ìa Ready
AND       U06.01.C	// _06_CH12_ACT ¨ú¨¡©ø?¡¤I¡¾¡¿AO¡¤A ¢¬©£¥ìa: A¢´©øI12 ¢¯iAuA©¬
AND       U06.18.C	// _06_CH12_IDD ¨ú¨¡©ø?¡¤I¡¾¡¿AO¡¤A ¢¬©£¥ìa: A¢´©øI12 AO¡¤A¢¥U¨ù¡¾¡ÆEAa
OR LOAD
AND       F0009A
OUT       M0087C	// R_2nd ALIGN ¢¥U¨ù¡¾¡ÆEAa
; L560
LOAD      M0087D	// R_3rd ALIGN ¢¥U¨ù¡¾¡ÆEAa
AND NOT   M00008	// LEFT RESET SW PLS
LOAD      U06.00.F	// _06_RDY ¨ú¨¡©ø?¡¤I¡¾¡¿AO¡¤A ¢¬©£¥ìa: ¢¬©£¥ìa Ready
AND       U06.01.D	// _06_CH13_ACT ¨ú¨¡©ø?¡¤I¡¾¡¿AO¡¤A ¢¬©£¥ìa: A¢´©øI13 ¢¯iAuA©¬
AND       U06.18.D	// _06_CH13_IDD ¨ú¨¡©ø?¡¤I¡¾¡¿AO¡¤A ¢¬©£¥ìa: A¢´©øI13 AO¡¤A¢¥U¨ù¡¾¡ÆEAa
OR LOAD
AND       F0009A
OUT       M0087D	// R_3rd ALIGN ¢¥U¨ù¡¾¡ÆEAa
; L562
LOAD      M0087E	// R_4th ALIGN ¢¥U¨ù¡¾¡ÆEAa
AND NOT   M00008	// LEFT RESET SW PLS
LOAD      U06.00.F	// _06_RDY ¨ú¨¡©ø?¡¤I¡¾¡¿AO¡¤A ¢¬©£¥ìa: ¢¬©£¥ìa Ready
AND       U06.01.E	// _06_CH14_ACT ¨ú¨¡©ø?¡¤I¡¾¡¿AO¡¤A ¢¬©£¥ìa: A¢´©øI14 ¢¯iAuA©¬
AND       U06.18.E	// _06_CH14_IDD ¨ú¨¡©ø?¡¤I¡¾¡¿AO¡¤A ¢¬©£¥ìa: A¢´©øI14 AO¡¤A¢¥U¨ù¡¾¡ÆEAa
OR LOAD
AND       F0009A
OUT       M0087E	// R_4th ALIGN ¢¥U¨ù¡¾¡ÆEAa

